LIN {X 0,Y 501.339,Z 1081.157,A -85,B 0,C 180,E1 23643.313,E2 23643.313} C_VEL
LIN {X 0,Y 503.042,Z 1063.83,A -85,B 0,C 180,E1 23641.19,E2 23641.19} C_VEL
LIN {X 0,Y 504.709,Z 1046.952,A -85,B 0,C 180,E1 23639.393,E2 23639.393} C_VEL
LIN {X 0,Y 506.659,Z 1027.452,A -85,B 0,C 180,E1 23637.597,E2 23637.597} C_VEL
LIN {X 0,Y 508.469,Z 1008.885,A -85,B 0,C 180,E1 23636.118,E2 23636.118} C_VEL
LIN {X 0,Y 510.36,Z 987.812,A -85,B 0,C 180,E1 23634.694,E2 23634.694} C_VEL
LIN {X 0,Y 512.134,Z 967.274,A -85,B 0,C 180,E1 23633.523,E2 23633.523} C_VEL
LIN {X 0,Y 513.653,Z 946.062,A -85,B 0,C 180,E1 23632.54,E2 23632.54} C_VEL
LIN {X 0,Y 515.046,Z 923.99,A -85,B 0,C 180,E1 23631.712,E2 23631.712} C_VEL
LIN {X 0,Y 516.104,Z 901.792,A -85,B 0,C 180,E1 23631.102,E2 23631.102} C_VEL
LIN {X 0,Y 516.884,Z 877.055,A -85,B 0,C 180,E1 23630.622,E2 23630.622} C_VEL
LIN {X 0,Y 520.36,Z 675.514,A -85,B 0,C 180,E1 23627.344,E2 23627.344} C_VEL
LIN {X 0,Y 522.211,Z 567.304,A -85,B 0,C 180,E1 23625.529,E2 23625.529} C_VEL
LIN {X 0,Y 521.353,Z 564.118,A -85,B 0,C 180,E1 23625.377,E2 23625.377} C_VEL
LIN {X 0,Y 506.181,Z 540.947,A -85,B 0,C 180,E1 23623.206,E2 23623.206} C_VEL
LIN {X 0,Y 500.368,Z 529.073,A -85,B 0,C 180,E1 23621.408,E2 23621.408} C_VEL
LIN {X 0,Y 498.57,Z 525.359,A -85,B 0,C 180,E1 23620.827,E2 23620.827} C_VEL
LIN {X 0,Y 496.912,Z 522.181,A -85,B 0,C 180,E1 23620.305,E2 23620.305} C_VEL
LIN {X 0,Y 496.727,Z 521.177,A -85,B 0,C 180,E1 23620.175,E2 23620.175} C_VEL
LIN {X 0,Y 496.731,Z 521.174,A -85,B 0,C 180,E1 23616.568,E2 23616.568} C_VEL
LIN {X 0,Y 496.77,Z 521.152,A -85,B 0,C 180,E1 23613.055,E2 23613.055} C_VEL
LIN {X 0,Y 496.742,Z 521.144,A -85,B 0,C 180,E1 23609.547,E2 23609.547} C_VEL
LIN {X 0,Y 496.741,Z 521.166,A -85,B 0,C 180,E1 23606.027,E2 23606.027} C_VEL
LIN {X 0,Y 496.765,Z 521.148,A -85,B 0,C 180,E1 23602.483,E2 23602.483} C_VEL
LIN {X 0,Y 496.759,Z 521.148,A -85,B 0,C 180,E1 23598.908,E2 23598.908} C_VEL
LIN {X 0,Y 496.747,Z 521.161,A -85,B 0,C 180,E1 23595.389,E2 23595.389} C_VEL
LIN {X 0,Y 496.76,Z 521.146,A -85,B 0,C 180,E1 23591.965,E2 23591.965} C_VEL
LIN {X 0,Y 496.766,Z 521.164,A -85,B 0,C 180,E1 23588.332,E2 23588.332} C_VEL
LIN {X 0,Y 496.756,Z 521.163,A -85,B 0,C 180,E1 23584.733,E2 23584.733} C_VEL
LIN {X 0,Y 496.765,Z 521.162,A -85,B 0,C 180,E1 23581.153,E2 23581.153} C_VEL
LIN {X 0,Y 496.749,Z 521.17,A -85,B 0,C 180,E1 23577.577,E2 23577.577} C_VEL
LIN {X 0,Y 496.767,Z 521.163,A -85,B 0,C 180,E1 23573.992,E2 23573.992} C_VEL
LIN {X 0,Y 496.764,Z 521.144,A -85,B 0,C 180,E1 23570.383,E2 23570.383} C_VEL
LIN {X 0,Y 496.739,Z 521.168,A -85,B 0,C 180,E1 23566.853,E2 23566.853} C_VEL
LIN {X 0,Y 496.756,Z 521.139,A -85,B 0,C 180,E1 23563.354,E2 23563.354} C_VEL
LIN {X 0,Y 496.765,Z 521.164,A -85,B 0,C 180,E1 23559.868,E2 23559.868} C_VEL
LIN {X 0,Y 496.722,Z 521.139,A -85,B 0,C 180,E1 23556.512,E2 23556.512} C_VEL
LIN {X 0,Y 496.769,Z 521.171,A -85,B 0,C 180,E1 23553.072,E2 23553.072} C_VEL
LIN {X 0,Y 496.728,Z 521.149,A -85,B 0,C 180,E1 23549.653,E2 23549.653} C_VEL
LIN {X 0,Y 496.717,Z 521.157,A -85,B 0,C 180,E1 23546.238,E2 23546.238} C_VEL
LIN {X 0,Y 496.767,Z 521.171,A -85,B 0,C 180,E1 23542.849,E2 23542.849} C_VEL
LIN {X 0,Y 496.704,Z 521.167,A -85,B 0,C 180,E1 23539.444,E2 23539.444} C_VEL
LIN {X 0,Y 496.719,Z 521.291,A -85,B 0,C 180,E1 23537.8,E2 23537.8} C_VEL
LIN {X 0,Y 497.882,Z 524.471,A -85,B 0,C 180,E1 23537.584,E2 23537.584} C_VEL
LIN {X 0,Y 500.714,Z 527.592,A -85,B 0,C 180,E1 23537.161,E2 23537.161} C_VEL
LIN {X 0,Y 503.416,Z 531.516,A -85,B 0,C 180,E1 23536.747,E2 23536.747} C_VEL
LIN {X 0,Y 515.125,Z 547.854,A -85,B 0,C 180,E1 23535.047,E2 23535.047} C_VEL
LIN {X 0,Y 522.101,Z 558.293,A -85,B 0,C 180,E1 23534.08,E2 23534.08} C_VEL
LIN {X 0,Y 521.82,Z 573.27,A -85,B 0,C 180,E1 23533.828,E2 23533.828} C_VEL
LIN {X 0,Y 520.938,Z 580.975,A -85,B 0,C 180,E1 23533.777,E2 23533.777} C_VEL
LIN {X 0,Y 516.065,Z 601.619,A -85,B 0,C 180,E1 23533.91,E2 23533.91} C_VEL
LIN {X 0,Y 515.408,Z 608.225,A -85,B 0,C 180,E1 23533.855,E2 23533.855} C_VEL
LIN {X 0,Y 511.275,Z 818.012,A -85,B 0,C 180,E1 23530.381,E2 23530.381} C_VEL
LIN {X 0,Y 510.22,Z 865.585,A -85,B 0,C 180,E1 23529.57,E2 23529.57} C_VEL
LIN {X 0,Y 509.144,Z 887.086,A -85,B 0,C 180,E1 23529.015,E2 23529.015} C_VEL
LIN {X 0,Y 507.847,Z 908.352,A -85,B 0,C 180,E1 23528.294,E2 23528.294} C_VEL
LIN {X 0,Y 506.128,Z 930.123,A -85,B 0,C 180,E1 23527.336,E2 23527.336} C_VEL
LIN {X 0,Y 504.269,Z 952.142,A -85,B 0,C 180,E1 23526.149,E2 23526.149} C_VEL
LIN {X 0,Y 502.401,Z 971.336,A -85,B 0,C 180,E1 23524.902,E2 23524.902} C_VEL
LIN {X 0,Y 500.276,Z 991.897,A -85,B 0,C 180,E1 23523.34,E2 23523.34} C_VEL
LIN {X 0,Y 498.327,Z 1010.198,A -85,B 0,C 180,E1 23521.709,E2 23521.709} C_VEL
LIN {X 0,Y 496.2,Z 1029.513,A -85,B 0,C 180,E1 23519.716,E2 23519.716} C_VEL
LIN {X 0,Y 494.437,Z 1046.319,A -85,B 0,C 180,E1 23517.718,E2 23517.718} C_VEL
LIN {X 0,Y 492.742,Z 1062.531,A -85,B 0,C 180,E1 23515.48,E2 23515.48} C_VEL
LIN {X 0,Y 491.262,Z 1078.098,A -85,B 0,C 180,E1 23513.003,E2 23513.003} C_VEL
LIN {X 0,Y 490.193,Z 1090.761,A -85,B 0,C 180,E1 23510.663,E2 23510.663} C_VEL
LIN {X 0,Y 489.317,Z 1102.656,A -85,B 0,C 180,E1 23508.095,E2 23508.095} C_VEL
LIN {X 0,Y 488.702,Z 1112.905,A -85,B 0,C 180,E1 23505.497,E2 23505.497} C_VEL
LIN {X 0,Y 488.285,Z 1121.274,A -85,B 0,C 180,E1 23502.897,E2 23502.897} C_VEL
LIN {X 0,Y 488.063,Z 1128.202,A -85,B 0,C 180,E1 23500.267,E2 23500.267} C_VEL
LIN {X 0,Y 487.966,Z 1133.176,A -85,B 0,C 180,E1 23497.773,E2 23497.773} C_VEL
LIN {X 0,Y 487.917,Z 1137.117,A -85,B 0,C 180,E1 23495.056,E2 23495.056} C_VEL
LIN {X 0,Y 487.91,Z 1139.232,A -85,B 0,C 180,E1 23492.467,E2 23492.467} C_VEL
LIN {X 0,Y 487.908,Z 1139.993,A -85,B 0,C 180,E1 23489.883,E2 23489.883} C_VEL
LIN {X 0,Y 487.904,Z 1139.148,A -85,B 0,C 180,E1 23487.299,E2 23487.299} C_VEL
LIN {X 0,Y 487.917,Z 1136.97,A -85,B 0,C 180,E1 23484.709,E2 23484.709} C_VEL
LIN {X 0,Y 487.97,Z 1133.127,A -85,B 0,C 180,E1 23482.109,E2 23482.109} C_VEL
LIN {X 0,Y 488.081,Z 1127.881,A -85,B 0,C 180,E1 23479.495,E2 23479.495} C_VEL
LIN {X 0,Y 488.313,Z 1120.835,A -85,B 0,C 180,E1 23476.863,E2 23476.863} C_VEL
LIN {X 0,Y 488.739,Z 1112.155,A -85,B 0,C 180,E1 23474.211,E2 23474.211} C_VEL
LIN {X 0,Y 489.361,Z 1102.001,A -85,B 0,C 180,E1 23471.66,E2 23471.66} C_VEL
LIN {X 0,Y 490.305,Z 1089.313,A -85,B 0,C 180,E1 23468.967,E2 23468.967} C_VEL
LIN {X 0,Y 491.452,Z 1076.174,A -85,B 0,C 180,E1 23466.572,E2 23466.572} C_VEL
LIN {X 0,Y 492.861,Z 1061.34,A -85,B 0,C 180,E1 23464.255,E2 23464.255} C_VEL
LIN {X 0,Y 494.567,Z 1044.991,A -85,B 0,C 180,E1 23462.029,E2 23462.029} C_VEL
LIN {X 0,Y 496.302,Z 1028.605,A -85,B 0,C 180,E1 23460.091,E2 23460.091} C_VEL
LIN {X 0,Y 498.378,Z 1009.706,A -85,B 0,C 180,E1 23458.154,E2 23458.154} C_VEL
LIN {X 0,Y 500.334,Z 991.393,A -85,B 0,C 180,E1 23456.526,E2 23456.526} C_VEL
LIN {X 0,Y 502.374,Z 971.61,A -85,B 0,C 180,E1 23455.027,E2 23455.027} C_VEL
LIN {X 0,Y 504.24,Z 952.427,A -85,B 0,C 180,E1 23453.779,E2 23453.779} C_VEL
LIN {X 0,Y 506.064,Z 930.957,A -85,B 0,C 180,E1 23452.615,E2 23452.615} C_VEL
LIN {X 0,Y 507.833,Z 908.532,A -85,B 0,C 180,E1 23451.623,E2 23451.623} C_VEL
LIN {X 0,Y 509.134,Z 887.292,A -85,B 0,C 180,E1 23450.901,E2 23450.901} C_VEL
LIN {X 0,Y 510.198,Z 866.05,A -85,B 0,C 180,E1 23450.351,E2 23450.351} C_VEL
LIN {X 0,Y 511.17,Z 823.523,A -85,B 0,C 180,E1 23449.619,E2 23449.619} C_VEL
LIN {X 0,Y 515.352,Z 611.14,A -85,B 0,C 180,E1 23446.104,E2 23446.104} C_VEL
LIN {X 0,Y 516.192,Z 561.548,A -85,B 0,C 180,E1 23445.247,E2 23445.247} C_VEL
LIN {X 0,Y 503.138,Z 542.859,A -85,B 0,C 180,E1 23443.361,E2 23443.361} C_VEL
LIN {X 0,Y 495.758,Z 532.811,A -85,B 0,C 180,E1 23442.23,E2 23442.23} C_VEL
LIN {X 0,Y 493.019,Z 529.057,A -85,B 0,C 180,E1 23441.795,E2 23441.795} C_VEL
LIN {X 0,Y 492.07,Z 527.668,A -85,B 0,C 180,E1 23441.64,E2 23441.64} C_VEL
LIN {X 0,Y 489.619,Z 524.782,A -85,B 0,C 180,E1 23441.25,E2 23441.25} C_VEL
LIN {X 0,Y 488.798,Z 522.162,A -85,B 0,C 180,E1 23441.07,E2 23441.07} C_VEL
LIN {X 0,Y 488.779,Z 522.154,A -85,B 0,C 180,E1 23437.708,E2 23437.708} C_VEL
LIN {X 0,Y 488.767,Z 522.136,A -85,B 0,C 180,E1 23434.233,E2 23434.233} C_VEL
LIN {X 0,Y 488.832,Z 522.142,A -85,B 0,C 180,E1 23430.754,E2 23430.754} C_VEL
LIN {X 0,Y 488.792,Z 522.155,A -85,B 0,C 180,E1 23427.272,E2 23427.272} C_VEL
LIN {X 0,Y 488.782,Z 522.128,A -85,B 0,C 180,E1 23423.765,E2 23423.765} C_VEL
LIN {X 0,Y 488.835,Z 522.157,A -85,B 0,C 180,E1 23420.348,E2 23420.348} C_VEL
LIN {X 0,Y 488.8,Z 522.124,A -85,B 0,C 180,E1 23416.801,E2 23416.801} C_VEL
LIN {X 0,Y 488.799,Z 522.158,A -85,B 0,C 180,E1 23413.244,E2 23413.244} C_VEL
LIN {X 0,Y 488.829,Z 522.155,A -85,B 0,C 180,E1 23409.775,E2 23409.775} C_VEL
LIN {X 0,Y 488.821,Z 522.161,A -85,B 0,C 180,E1 23406.224,E2 23406.224} C_VEL
LIN {X 0,Y 488.806,Z 522.159,A -85,B 0,C 180,E1 23402.58,E2 23402.58} C_VEL
LIN {X 0,Y 488.829,Z 522.154,A -85,B 0,C 180,E1 23399.063,E2 23399.063} C_VEL
LIN {X 0,Y 488.822,Z 522.157,A -85,B 0,C 180,E1 23395.425,E2 23395.425} C_VEL
LIN {X 0,Y 488.819,Z 522.159,A -85,B 0,C 180,E1 23391.887,E2 23391.887} C_VEL
LIN {X 0,Y 488.823,Z 522.122,A -85,B 0,C 180,E1 23388.317,E2 23388.317} C_VEL
LIN {X 0,Y 488.811,Z 522.155,A -85,B 0,C 180,E1 23384.822,E2 23384.822} C_VEL
LIN {X 0,Y 488.825,Z 522.13,A -85,B 0,C 180,E1 23381.269,E2 23381.269} C_VEL
LIN {X 0,Y 488.83,Z 522.144,A -85,B 0,C 180,E1 23377.639,E2 23377.639} C_VEL
LIN {X 0,Y 488.803,Z 522.159,A -85,B 0,C 180,E1 23374.04,E2 23374.04} C_VEL
LIN {X 0,Y 488.802,Z 522.135,A -85,B 0,C 180,E1 23370.383,E2 23370.383} C_VEL
LIN {X 0,Y 488.831,Z 522.137,A -85,B 0,C 180,E1 23366.899,E2 23366.899} C_VEL
LIN {X 0,Y 488.792,Z 522.161,A -85,B 0,C 180,E1 23363.469,E2 23363.469} C_VEL
LIN {X 0,Y 488.861,Z 522.355,A -85,B 0,C 180,E1 23360.759,E2 23360.759} C_VEL
LIN {X 0,Y 490.363,Z 525.981,A -85,B 0,C 180,E1 23360.19,E2 23360.19} C_VEL
LIN {X 0,Y 491.426,Z 528.1,A -85,B 0,C 180,E1 23359.837,E2 23359.837} C_VEL
LIN {X 0,Y 495.467,Z 535.911,A -85,B 0,C 180,E1 23358.555,E2 23358.555} C_VEL
LIN {X 0,Y 498.071,Z 541.152,A -85,B 0,C 180,E1 23357.783,E2 23357.783} C_VEL
LIN {X 0,Y 511.268,Z 561.075,A -85,B 0,C 180,E1 23355.799,E2 23355.799} C_VEL
LIN {X 0,Y 516.559,Z 569.744,A -85,B 0,C 180,E1 23355.037,E2 23355.037} C_VEL
LIN {X 0,Y 513.282,Z 735.937,A -85,B 0,C 180,E1 23352.257,E2 23352.257} C_VEL
LIN {X 0,Y 510.262,Z 891.967,A -85,B 0,C 180,E1 23349.679,E2 23349.679} C_VEL
LIN {X 0,Y 509.215,Z 914.865,A -85,B 0,C 180,E1 23349.119,E2 23349.119} C_VEL
LIN {X 0,Y 508.04,Z 934.757,A -85,B 0,C 180,E1 23348.465,E2 23348.465} C_VEL
LIN {X 0,Y 506.385,Z 957.093,A -85,B 0,C 180,E1 23347.527,E2 23347.527} C_VEL
LIN {X 0,Y 504.587,Z 978.468,A -85,B 0,C 180,E1 23346.411,E2 23346.411} C_VEL
LIN {X 0,Y 502.614,Z 999.226,A -85,B 0,C 180,E1 23345.093,E2 23345.093} C_VEL
LIN {X 0,Y 500.642,Z 1018.623,A -85,B 0,C 180,E1 23343.656,E2 23343.656} C_VEL
LIN {X 0,Y 498.56,Z 1037.927,A -85,B 0,C 180,E1 23341.968,E2 23341.968} C_VEL
LIN {X 0,Y 496.548,Z 1056.565,A -85,B 0,C 180,E1 23340.092,E2 23340.092} C_VEL
LIN {X 0,Y 494.748,Z 1073.124,A -85,B 0,C 180,E1 23338.157,E2 23338.157} C_VEL
LIN {X 0,Y 492.965,Z 1090.295,A -85,B 0,C 180,E1 23335.854,E2 23335.854} C_VEL
LIN {X 0,Y 491.518,Z 1105.507,A -85,B 0,C 180,E1 23333.497,E2 23333.497} C_VEL
LIN {X 0,Y 490.322,Z 1119.085,A -85,B 0,C 180,E1 23331.032,E2 23331.032} C_VEL
LIN {X 0,Y 489.407,Z 1131.29,A -85,B 0,C 180,E1 23328.461,E2 23328.461} C_VEL
LIN {X 0,Y 488.785,Z 1141.067,A -85,B 0,C 180,E1 23326.031,E2 23326.031} C_VEL
LIN {X 0,Y 488.334,Z 1150.349,A -85,B 0,C 180,E1 23323.257,E2 23323.257} C_VEL
LIN {X 0,Y 488.107,Z 1157.169,A -85,B 0,C 180,E1 23320.743,E2 23320.743} C_VEL
LIN {X 0,Y 487.975,Z 1162.635,A -85,B 0,C 180,E1 23318.128,E2 23318.128} C_VEL
LIN {X 0,Y 487.906,Z 1166.438,A -85,B 0,C 180,E1 23315.645,E2 23315.645} C_VEL
LIN {X 0,Y 487.89,Z 1168.986,A -85,B 0,C 180,E1 23312.937,E2 23312.937} C_VEL
LIN {X 0,Y 487.885,Z 1169.895,A -85,B 0,C 180,E1 23310.587,E2 23310.587} C_VEL
LIN {X 0,Y 487.914,Z 1169.392,A -85,B 0,C 180,E1 23307.768,E2 23307.768} C_VEL
LIN {X 0,Y 487.909,Z 1167.501,A -85,B 0,C 180,E1 23305.298,E2 23305.298} C_VEL
LIN {X 0,Y 487.933,Z 1163.874,A -85,B 0,C 180,E1 23302.582,E2 23302.582} C_VEL
LIN {X 0,Y 488.014,Z 1159.573,A -85,B 0,C 180,E1 23300.328,E2 23300.328} C_VEL
LIN {X 0,Y 488.213,Z 1153.516,A -85,B 0,C 180,E1 23297.822,E2 23297.822} C_VEL
LIN {X 0,Y 488.562,Z 1145.341,A -85,B 0,C 180,E1 23295.178,E2 23295.178} C_VEL
LIN {X 0,Y 489.13,Z 1135.417,A -85,B 0,C 180,E1 23292.513,E2 23292.513} C_VEL
LIN {X 0,Y 489.891,Z 1124.575,A -85,B 0,C 180,E1 23290.071,E2 23290.071} C_VEL
LIN {X 0,Y 490.992,Z 1111.15,A -85,B 0,C 180,E1 23287.49,E2 23287.49} C_VEL
LIN {X 0,Y 492.316,Z 1097.011,A -85,B 0,C 180,E1 23285.14,E2 23285.14} C_VEL
LIN {X 0,Y 493.871,Z 1081.33,A -85,B 0,C 180,E1 23282.901,E2 23282.901} C_VEL
LIN {X 0,Y 495.764,Z 1063.774,A -85,B 0,C 180,E1 23280.72,E2 23280.72} C_VEL
LIN {X 0,Y 497.616,Z 1046.551,A -85,B 0,C 180,E1 23278.865,E2 23278.865} C_VEL
LIN {X 0,Y 499.765,Z 1026.775,A -85,B 0,C 180,E1 23277.031,E2 23277.031} C_VEL
LIN {X 0,Y 501.819,Z 1007.26,A -85,B 0,C 180,E1 23275.468,E2 23275.468} C_VEL
LIN {X 0,Y 503.804,Z 986.803,A -85,B 0,C 180,E1 23274.094,E2 23274.094} C_VEL
LIN {X 0,Y 505.708,Z 966.071,A -85,B 0,C 180,E1 23272.912,E2 23272.912} C_VEL
LIN {X 0,Y 507.292,Z 945.156,A -85,B 0,C 180,E1 23271.944,E2 23271.944} C_VEL
LIN {X 0,Y 508.798,Z 922.523,A -85,B 0,C 180,E1 23271.108,E2 23271.108} C_VEL
LIN {X 0,Y 509.869,Z 901.392,A -85,B 0,C 180,E1 23270.529,E2 23270.529} C_VEL
LIN {X 0,Y 510.697,Z 876.242,A -85,B 0,C 180,E1 23270.041,E2 23270.041} C_VEL
LIN {X 0,Y 514.468,Z 675.084,A -85,B 0,C 180,E1 23266.734,E2 23266.734} C_VEL
LIN {X 0,Y 516.46,Z 569.215,A -85,B 0,C 180,E1 23264.942,E2 23264.942} C_VEL
LIN {X 0,Y 501.454,Z 546.105,A -85,B 0,C 180,E1 23262.74,E2 23262.74} C_VEL
LIN {X 0,Y 497.653,Z 540.451,A -85,B 0,C 180,E1 23262.148,E2 23262.148} C_VEL
LIN {X 0,Y 492.496,Z 530.229,A -85,B 0,C 180,E1 23260.515,E2 23260.515} C_VEL
LIN {X 0,Y 490.353,Z 525.974,A -85,B 0,C 180,E1 23259.811,E2 23259.811} C_VEL
LIN {X 0,Y 488.857,Z 522.324,A -85,B 0,C 180,E1 23259.241,E2 23259.241} C_VEL
LIN {X 0,Y 488.808,Z 522.153,A -85,B 0,C 180,E1 23255.701,E2 23255.701} C_VEL
LIN {X 0,Y 488.791,Z 522.159,A -85,B 0,C 180,E1 23252.126,E2 23252.126} C_VEL
LIN {X 0,Y 488.829,Z 522.13,A -85,B 0,C 180,E1 23248.595,E2 23248.595} C_VEL
LIN {X 0,Y 488.825,Z 522.135,A -85,B 0,C 180,E1 23245.023,E2 23245.023} C_VEL
LIN {X 0,Y 488.803,Z 522.152,A -85,B 0,C 180,E1 23241.452,E2 23241.452} C_VEL
LIN {X 0,Y 488.818,Z 522.121,A -85,B 0,C 180,E1 23237.867,E2 23237.867} C_VEL
LIN {X 0,Y 488.825,Z 522.159,A -85,B 0,C 180,E1 23234.329,E2 23234.329} C_VEL
LIN {X 0,Y 488.816,Z 522.123,A -85,B 0,C 180,E1 23230.727,E2 23230.727} C_VEL
LIN {X 0,Y 488.822,Z 522.156,A -85,B 0,C 180,E1 23227.167,E2 23227.167} C_VEL
LIN {X 0,Y 488.815,Z 522.157,A -85,B 0,C 180,E1 23223.635,E2 23223.635} C_VEL
LIN {X 0,Y 488.827,Z 522.159,A -85,B 0,C 180,E1 23220,E2 23220} C_VEL
LIN {X 0,Y 488.824,Z 522.158,A -85,B 0,C 180,E1 23216.364,E2 23216.364} C_VEL
LIN {X 0,Y 488.825,Z 522.155,A -85,B 0,C 180,E1 23212.714,E2 23212.714} C_VEL
LIN {X 0,Y 488.798,Z 522.125,A -85,B 0,C 180,E1 23209.074,E2 23209.074} C_VEL
LIN {X 0,Y 488.832,Z 522.158,A -85,B 0,C 180,E1 23205.55,E2 23205.55} C_VEL
LIN {X 0,Y 488.827,Z 522.122,A -85,B 0,C 180,E1 23201.886,E2 23201.886} C_VEL
LIN {X 0,Y 488.792,Z 522.156,A -85,B 0,C 180,E1 23198.395,E2 23198.395} C_VEL
LIN {X 0,Y 488.799,Z 522.14,A -85,B 0,C 180,E1 23194.819,E2 23194.819} C_VEL
LIN {X 0,Y 488.834,Z 522.134,A -85,B 0,C 180,E1 23191.34,E2 23191.34} C_VEL
LIN {X 0,Y 488.779,Z 522.162,A -85,B 0,C 180,E1 23187.868,E2 23187.868} C_VEL
LIN {X 0,Y 488.783,Z 522.143,A -85,B 0,C 180,E1 23184.303,E2 23184.303} C_VEL
LIN {X 0,Y 488.809,Z 522.134,A -85,B 0,C 180,E1 23180.949,E2 23180.949} C_VEL
LIN {X 0,Y 488.831,Z 522.299,A -85,B 0,C 180,E1 23178.818,E2 23178.818} C_VEL
LIN {X 0,Y 490.064,Z 525.535,A -85,B 0,C 180,E1 23178.581,E2 23178.581} C_VEL
LIN {X 0,Y 492.832,Z 528.661,A -85,B 0,C 180,E1 23178.147,E2 23178.147} C_VEL
LIN {X 0,Y 495.553,Z 532.605,A -85,B 0,C 180,E1 23177.709,E2 23177.709} C_VEL
LIN {X 0,Y 497.132,Z 534.605,A -85,B 0,C 180,E1 23177.465,E2 23177.465} C_VEL
LIN {X 0,Y 510.465,Z 553.132,A -85,B 0,C 180,E1 23175.475,E2 23175.475} C_VEL
LIN {X 0,Y 516.314,Z 562.022,A -85,B 0,C 180,E1 23174.64,E2 23174.64} C_VEL
LIN {X 0,Y 515.408,Z 608.225,A -85,B 0,C 180,E1 23173.855,E2 23173.855} C_VEL
LIN {X 0,Y 514.536,Z 615.928,A -85,B 0,C 180,E1 23173.803,E2 23173.803} C_VEL
LIN {X 0,Y 509.557,Z 636.554,A -85,B 0,C 180,E1 23173.949,E2 23173.949} C_VEL
LIN {X 0,Y 508.877,Z 643.162,A -85,B 0,C 180,E1 23173.896,E2 23173.896} C_VEL
LIN {X 0,Y 504.713,Z 842.961,A -85,B 0,C 180,E1 23170.563,E2 23170.563} C_VEL
LIN {X 0,Y 503.803,Z 871.088,A -85,B 0,C 180,E1 23170.027,E2 23170.027} C_VEL
LIN {X 0,Y 502.74,Z 890.849,A -85,B 0,C 180,E1 23169.487,E2 23169.487} C_VEL
LIN {X 0,Y 501.099,Z 913.862,A -85,B 0,C 180,E1 23168.649,E2 23168.649} C_VEL
LIN {X 0,Y 499.365,Z 934.763,A -85,B 0,C 180,E1 23167.68,E2 23167.68} C_VEL
LIN {X 0,Y 497.285,Z 956.054,A -85,B 0,C 180,E1 23166.462,E2 23166.462} C_VEL
LIN {X 0,Y 495.126,Z 976.727,A -85,B 0,C 180,E1 23165.067,E2 23165.067} C_VEL
LIN {X 0,Y 492.895,Z 996.298,A -85,B 0,C 180,E1 23163.489,E2 23163.489} C_VEL
LIN {X 0,Y 490.692,Z 1015.331,A -85,B 0,C 180,E1 23161.717,E2 23161.717} C_VEL
LIN {X 0,Y 488.602,Z 1032.911,A -85,B 0,C 180,E1 23159.812,E2 23159.812} C_VEL
LIN {X 0,Y 486.55,Z 1050.552,A -85,B 0,C 180,E1 23157.607,E2 23157.607} C_VEL
LIN {X 0,Y 484.884,Z 1065.915,A -85,B 0,C 180,E1 23155.399,E2 23155.399} C_VEL
LIN {X 0,Y 483.397,Z 1080.22,A -85,B 0,C 180,E1 23153.009,E2 23153.009} C_VEL
LIN {X 0,Y 482.221,Z 1093.21,A -85,B 0,C 180,E1 23150.513,E2 23150.513} C_VEL
LIN {X 0,Y 481.354,Z 1104.202,A -85,B 0,C 180,E1 23148.029,E2 23148.029} C_VEL
LIN {X 0,Y 480.667,Z 1114.787,A -85,B 0,C 180,E1 23145.195,E2 23145.195} C_VEL
LIN {X 0,Y 480.268,Z 1122.688,A -85,B 0,C 180,E1 23142.627,E2 23142.627} C_VEL
LIN {X 0,Y 480.035,Z 1129.224,A -85,B 0,C 180,E1 23139.956,E2 23139.956} C_VEL
LIN {X 0,Y 479.957,Z 1133.59,A -85,B 0,C 180,E1 23137.662,E2 23137.662} C_VEL
LIN {X 0,Y 479.915,Z 1137.344,A -85,B 0,C 180,E1 23134.9,E2 23134.9} C_VEL
LIN {X 0,Y 479.912,Z 1139.3,A -85,B 0,C 180,E1 23132.388,E2 23132.388} C_VEL
LIN {X 0,Y 479.892,Z 1139.948,A -85,B 0,C 180,E1 23129.642,E2 23129.642} C_VEL
LIN {X 0,Y 479.902,Z 1139.148,A -85,B 0,C 180,E1 23127.254,E2 23127.254} C_VEL
LIN {X 0,Y 479.917,Z 1136.969,A -85,B 0,C 180,E1 23124.621,E2 23124.621} C_VEL
LIN {X 0,Y 479.978,Z 1133.126,A -85,B 0,C 180,E1 23121.977,E2 23121.977} C_VEL
LIN {X 0,Y 480.107,Z 1127.879,A -85,B 0,C 180,E1 23119.319,E2 23119.319} C_VEL
LIN {X 0,Y 480.362,Z 1120.832,A -85,B 0,C 180,E1 23116.642,E2 23116.642} C_VEL
LIN {X 0,Y 480.825,Z 1112.15,A -85,B 0,C 180,E1 23113.945,E2 23113.945} C_VEL
LIN {X 0,Y 481.477,Z 1102.511,A -85,B 0,C 180,E1 23111.475,E2 23111.475} C_VEL
LIN {X 0,Y 482.503,Z 1089.942,A -85,B 0,C 180,E1 23108.738,E2 23108.738} C_VEL
LIN {X 0,Y 483.71,Z 1077.184,A -85,B 0,C 180,E1 23106.359,E2 23106.359} C_VEL
LIN {X 0,Y 485.274,Z 1062.091,A -85,B 0,C 180,E1 23103.94,E2 23103.94} C_VEL
LIN {X 0,Y 487.11,Z 1045.998,A -85,B 0,C 180,E1 23101.696,E2 23101.696} C_VEL
LIN {X 0,Y 489.041,Z 1029.151,A -85,B 0,C 180,E1 23099.669,E2 23099.669} C_VEL
LIN {X 0,Y 491.379,Z 1009.372,A -85,B 0,C 180,E1 23097.612,E2 23097.612} C_VEL
LIN {X 0,Y 493.524,Z 990.907,A -85,B 0,C 180,E1 23095.957,E2 23095.957} C_VEL
LIN {X 0,Y 495.758,Z 970.694,A -85,B 0,C 180,E1 23094.419,E2 23094.419} C_VEL
LIN {X 0,Y 497.881,Z 950.461,A -85,B 0,C 180,E1 23093.097,E2 23093.097} C_VEL
LIN {X 0,Y 499.808,Z 929.406,A -85,B 0,C 180,E1 23091.965,E2 23091.965} C_VEL
LIN {X 0,Y 501.666,Z 907.09,A -85,B 0,C 180,E1 23090.989,E2 23090.989} C_VEL
LIN {X 0,Y 502.975,Z 886.817,A -85,B 0,C 180,E1 23090.302,E2 23090.302} C_VEL
LIN {X 0,Y 504.111,Z 865.028,A -85,B 0,C 180,E1 23089.742,E2 23089.742} C_VEL
LIN {X 0,Y 505.544,Z 801.78,A -85,B 0,C 180,E1 23088.667,E2 23088.667} C_VEL
LIN {X 0,Y 510.059,Z 589.597,A -85,B 0,C 180,E1 23085.106,E2 23085.106} C_VEL
LIN {X 0,Y 510.416,Z 565.256,A -85,B 0,C 180,E1 23084.669,E2 23084.669} C_VEL
LIN {X 0,Y 498.717,Z 548.51,A -85,B 0,C 180,E1 23082.934,E2 23082.934} C_VEL
LIN {X 0,Y 491.702,Z 538.917,A -85,B 0,C 180,E1 23081.834,E2 23081.834} C_VEL
LIN {X 0,Y 487.888,Z 533.76,A -85,B 0,C 180,E1 23081.214,E2 23081.214} C_VEL
LIN {X 0,Y 485.077,Z 529.758,A -85,B 0,C 180,E1 23080.741,E2 23080.741} C_VEL
LIN {X 0,Y 483.973,Z 528.567,A -85,B 0,C 180,E1 23080.561,E2 23080.561} C_VEL
LIN {X 0,Y 481.652,Z 525.825,A -85,B 0,C 180,E1 23080.172,E2 23080.172} C_VEL
LIN {X 0,Y 480.826,Z 523.131,A -85,B 0,C 180,E1 23079.983,E2 23079.983} C_VEL
LIN {X 0,Y 480.829,Z 523.152,A -85,B 0,C 180,E1 23076.345,E2 23076.345} C_VEL
LIN {X 0,Y 480.885,Z 523.137,A -85,B 0,C 180,E1 23072.86,E2 23072.86} C_VEL
LIN {X 0,Y 480.846,Z 523.119,A -85,B 0,C 180,E1 23069.389,E2 23069.389} C_VEL
LIN {X 0,Y 480.843,Z 523.149,A -85,B 0,C 180,E1 23065.76,E2 23065.76} C_VEL
LIN {X 0,Y 480.89,Z 523.122,A -85,B 0,C 180,E1 23062.236,E2 23062.236} C_VEL
LIN {X 0,Y 480.876,Z 523.128,A -85,B 0,C 180,E1 23058.675,E2 23058.675} C_VEL
LIN {X 0,Y 480.853,Z 523.138,A -85,B 0,C 180,E1 23055.065,E2 23055.065} C_VEL
LIN {X 0,Y 480.88,Z 523.14,A -85,B 0,C 180,E1 23051.514,E2 23051.514} C_VEL
LIN {X 0,Y 480.89,Z 523.14,A -85,B 0,C 180,E1 23047.888,E2 23047.888} C_VEL
LIN {X 0,Y 480.873,Z 523.14,A -85,B 0,C 180,E1 23044.293,E2 23044.293} C_VEL
LIN {X 0,Y 480.874,Z 523.136,A -85,B 0,C 180,E1 23040.715,E2 23040.715} C_VEL
LIN {X 0,Y 480.883,Z 523.139,A -85,B 0,C 180,E1 23037.14,E2 23037.14} C_VEL
LIN {X 0,Y 480.886,Z 523.14,A -85,B 0,C 180,E1 23033.434,E2 23033.434} C_VEL
LIN {X 0,Y 480.878,Z 523.118,A -85,B 0,C 180,E1 23029.821,E2 23029.821} C_VEL
LIN {X 0,Y 480.892,Z 523.141,A -85,B 0,C 180,E1 23026.162,E2 23026.162} C_VEL
LIN {X 0,Y 480.866,Z 523.112,A -85,B 0,C 180,E1 23022.578,E2 23022.578} C_VEL
LIN {X 0,Y 480.884,Z 523.148,A -85,B 0,C 180,E1 23018.918,E2 23018.918} C_VEL
LIN {X 0,Y 480.888,Z 523.121,A -85,B 0,C 180,E1 23015.297,E2 23015.297} C_VEL
LIN {X 0,Y 480.869,Z 523.126,A -85,B 0,C 180,E1 23011.701,E2 23011.701} C_VEL
LIN {X 0,Y 480.856,Z 523.149,A -85,B 0,C 180,E1 23008.12,E2 23008.12} C_VEL
LIN {X 0,Y 480.884,Z 523.135,A -85,B 0,C 180,E1 23004.543,E2 23004.543} C_VEL
LIN {X 0,Y 480.846,Z 523.131,A -85,B 0,C 180,E1 23001.814,E2 23001.814} C_VEL
LIN {X 0,Y 481.866,Z 526.149,A -85,B 0,C 180,E1 23001.35,E2 23001.35} C_VEL
LIN {X 0,Y 483.39,Z 528.554,A -85,B 0,C 180,E1 23000.886,E2 23000.886} C_VEL
LIN {X 0,Y 489.618,Z 540.648,A -85,B 0,C 180,E1 22998.886,E2 22998.886} C_VEL
LIN {X 0,Y 504.715,Z 563.364,A -85,B 0,C 180,E1 22996.516,E2 22996.516} C_VEL
LIN {X 0,Y 510.835,Z 573.306,A -85,B 0,C 180,E1 22995.608,E2 22995.608} C_VEL
LIN {X 0,Y 506.828,Z 762.387,A -85,B 0,C 180,E1 22992.42,E2 22992.42} C_VEL
LIN {X 0,Y 504.081,Z 891.906,A -85,B 0,C 180,E1 22990.259,E2 22990.259} C_VEL
LIN {X 0,Y 502.95,Z 914.763,A -85,B 0,C 180,E1 22989.694,E2 22989.694} C_VEL
LIN {X 0,Y 501.656,Z 935.178,A -85,B 0,C 180,E1 22989.016,E2 22989.016} C_VEL
LIN {X 0,Y 499.821,Z 958.146,A -85,B 0,C 180,E1 22988.034,E2 22988.034} C_VEL
LIN {X 0,Y 497.919,Z 979.647,A -85,B 0,C 180,E1 22986.9,E2 22986.9} C_VEL
LIN {X 0,Y 495.819,Z 1000.123,A -85,B 0,C 180,E1 22985.576,E2 22985.576} C_VEL
LIN {X 0,Y 493.621,Z 1020.17,A -85,B 0,C 180,E1 22984.061,E2 22984.061} C_VEL
LIN {X 0,Y 491.391,Z 1039.26,A -85,B 0,C 180,E1 22982.353,E2 22982.353} C_VEL
LIN {X 0,Y 489.088,Z 1058.783,A -85,B 0,C 180,E1 22980.328,E2 22980.328} C_VEL
LIN {X 0,Y 487.195,Z 1075.15,A -85,B 0,C 180,E1 22978.366,E2 22978.366} C_VEL
LIN {X 0,Y 485.378,Z 1091.139,A -85,B 0,C 180,E1 22976.157,E2 22976.157} C_VEL
LIN {X 0,Y 483.813,Z 1106.228,A -85,B 0,C 180,E1 22973.765,E2 22973.765} C_VEL
LIN {X 0,Y 482.57,Z 1119.083,A -85,B 0,C 180,E1 22971.387,E2 22971.387} C_VEL
LIN {X 0,Y 481.56,Z 1131.291,A -85,B 0,C 180,E1 22968.773,E2 22968.773} C_VEL
LIN {X 0,Y 480.878,Z 1141.066,A -85,B 0,C 180,E1 22966.302,E2 22966.302} C_VEL
LIN {X 0,Y 480.379,Z 1150.349,A -85,B 0,C 180,E1 22963.48,E2 22963.48} C_VEL
LIN {X 0,Y 480.127,Z 1157.169,A -85,B 0,C 180,E1 22960.924,E2 22960.924} C_VEL
LIN {X 0,Y 479.98,Z 1162.635,A -85,B 0,C 180,E1 22958.264,E2 22958.264} C_VEL
LIN {X 0,Y 479.907,Z 1166.438,A -85,B 0,C 180,E1 22955.739,E2 22955.739} C_VEL
LIN {X 0,Y 479.889,Z 1168.986,A -85,B 0,C 180,E1 22952.986,E2 22952.986} C_VEL
LIN {X 0,Y 479.884,Z 1169.895,A -85,B 0,C 180,E1 22950.597,E2 22950.597} C_VEL
LIN {X 0,Y 479.914,Z 1169.392,A -85,B 0,C 180,E1 22947.731,E2 22947.731} C_VEL
LIN {X 0,Y 479.91,Z 1167.501,A -85,B 0,C 180,E1 22945.219,E2 22945.219} C_VEL
LIN {X 0,Y 479.943,Z 1163.874,A -85,B 0,C 180,E1 22942.458,E2 22942.458} C_VEL
LIN {X 0,Y 480.028,Z 1159.507,A -85,B 0,C 180,E1 22940.134,E2 22940.134} C_VEL
LIN {X 0,Y 480.255,Z 1153.171,A -85,B 0,C 180,E1 22937.495,E2 22937.495} C_VEL
LIN {X 0,Y 480.636,Z 1145.34,A -85,B 0,C 180,E1 22934.927,E2 22934.927} C_VEL
LIN {X 0,Y 481.267,Z 1135.416,A -85,B 0,C 180,E1 22932.217,E2 22932.217} C_VEL
LIN {X 0,Y 482.101,Z 1124.575,A -85,B 0,C 180,E1 22929.735,E2 22929.735} C_VEL
LIN {X 0,Y 483.31,Z 1111.148,A -85,B 0,C 180,E1 22927.112,E2 22927.112} C_VEL
LIN {X 0,Y 484.765,Z 1097.013,A -85,B 0,C 180,E1 22924.725,E2 22924.725} C_VEL
LIN {X 0,Y 486.457,Z 1081.328,A -85,B 0,C 180,E1 22922.453,E2 22922.453} C_VEL
LIN {X 0,Y 488.452,Z 1064.328,A -85,B 0,C 180,E1 22920.305,E2 22920.305} C_VEL
LIN {X 0,Y 490.425,Z 1047.391,A -85,B 0,C 180,E1 22918.451,E2 22918.451} C_VEL
LIN {X 0,Y 492.764,Z 1027.507,A -85,B 0,C 180,E1 22916.571,E2 22916.571} C_VEL
LIN {X 0,Y 494.864,Z 1008.879,A -85,B 0,C 180,E1 22915.053,E2 22915.053} C_VEL
LIN {X 0,Y 496.993,Z 988.81,A -85,B 0,C 180,E1 22913.666,E2 22913.666} C_VEL
LIN {X 0,Y 498.886,Z 969.272,A -85,B 0,C 180,E1 22912.528,E2 22912.528} C_VEL
LIN {X 0,Y 500.735,Z 947.084,A -85,B 0,C 180,E1 22911.464,E2 22911.464} C_VEL
LIN {X 0,Y 502.305,Z 925.39,A -85,B 0,C 180,E1 22910.631,E2 22910.631} C_VEL
LIN {X 0,Y 503.58,Z 902.883,A -85,B 0,C 180,E1 22909.989,E2 22909.989} C_VEL
LIN {X 0,Y 504.483,Z 879.641,A -85,B 0,C 180,E1 22909.515,E2 22909.515} C_VEL
LIN {X 0,Y 508.542,Z 678.812,A -85,B 0,C 180,E1 22906.179,E2 22906.179} C_VEL
LIN {X 0,Y 510.672,Z 572.789,A -85,B 0,C 180,E1 22904.363,E2 22904.363} C_VEL
LIN {X 0,Y 496.157,Z 550.277,A -85,B 0,C 180,E1 22902.168,E2 22902.168} C_VEL
LIN {X 0,Y 489.059,Z 539.882,A -85,B 0,C 180,E1 22901.015,E2 22901.015} C_VEL
LIN {X 0,Y 484.254,Z 530.592,A -85,B 0,C 180,E1 22899.446,E2 22899.446} C_VEL
LIN {X 0,Y 483.081,Z 527.74,A -85,B 0,C 180,E1 22898.991,E2 22898.991} C_VEL
LIN {X 0,Y 481.2,Z 524.712,A -85,B 0,C 180,E1 22898.409,E2 22898.409} C_VEL
LIN {X 0,Y 480.848,Z 523.154,A -85,B 0,C 180,E1 22898.186,E2 22898.186} C_VEL
LIN {X 0,Y 480.859,Z 523.122,A -85,B 0,C 180,E1 22894.571,E2 22894.571} C_VEL
LIN {X 0,Y 480.894,Z 523.138,A -85,B 0,C 180,E1 22891.039,E2 22891.039} C_VEL
LIN {X 0,Y 480.866,Z 523.136,A -85,B 0,C 180,E1 22887.49,E2 22887.49} C_VEL
LIN {X 0,Y 480.862,Z 523.111,A -85,B 0,C 180,E1 22883.92,E2 22883.92} C_VEL
LIN {X 0,Y 480.89,Z 523.143,A -85,B 0,C 180,E1 22880.444,E2 22880.444} C_VEL
LIN {X 0,Y 480.883,Z 523.111,A -85,B 0,C 180,E1 22876.798,E2 22876.798} C_VEL
LIN {X 0,Y 480.874,Z 523.146,A -85,B 0,C 180,E1 22873.221,E2 22873.221} C_VEL
LIN {X 0,Y 480.886,Z 523.122,A -85,B 0,C 180,E1 22869.575,E2 22869.575} C_VEL
LIN {X 0,Y 480.879,Z 523.138,A -85,B 0,C 180,E1 22865.967,E2 22865.967} C_VEL
LIN {X 0,Y 480.884,Z 523.141,A -85,B 0,C 180,E1 22862.383,E2 22862.383} C_VEL
LIN {X 0,Y 480.888,Z 523.14,A -85,B 0,C 180,E1 22858.689,E2 22858.689} C_VEL
LIN {X 0,Y 480.871,Z 523.137,A -85,B 0,C 180,E1 22855.109,E2 22855.109} C_VEL
LIN {X 0,Y 480.874,Z 523.135,A -85,B 0,C 180,E1 22851.51,E2 22851.51} C_VEL
LIN {X 0,Y 480.89,Z 523.122,A -85,B 0,C 180,E1 22847.878,E2 22847.878} C_VEL
LIN {X 0,Y 480.877,Z 523.135,A -85,B 0,C 180,E1 22844.302,E2 22844.302} C_VEL
LIN {X 0,Y 480.853,Z 523.137,A -85,B 0,C 180,E1 22840.694,E2 22840.694} C_VEL
LIN {X 0,Y 480.878,Z 523.116,A -85,B 0,C 180,E1 22837.119,E2 22837.119} C_VEL
LIN {X 0,Y 480.882,Z 523.144,A -85,B 0,C 180,E1 22833.58,E2 22833.58} C_VEL
LIN {X 0,Y 480.836,Z 523.12,A -85,B 0,C 180,E1 22830.126,E2 22830.126} C_VEL
LIN {X 0,Y 480.861,Z 523.134,A -85,B 0,C 180,E1 22826.563,E2 22826.563} C_VEL
LIN {X 0,Y 480.873,Z 523.149,A -85,B 0,C 180,E1 22823.065,E2 22823.065} C_VEL
LIN {X 0,Y 480.85,Z 523.298,A -85,B 0,C 180,E1 22819.906,E2 22819.906} C_VEL
LIN {X 0,Y 482.011,Z 526.442,A -85,B 0,C 180,E1 22819.669,E2 22819.669} C_VEL
LIN {X 0,Y 484.677,Z 529.028,A -85,B 0,C 180,E1 22819.238,E2 22819.238} C_VEL
LIN {X 0,Y 487.533,Z 533.4,A -85,B 0,C 180,E1 22818.75,E2 22818.75} C_VEL
LIN {X 0,Y 489.227,Z 535.532,A -85,B 0,C 180,E1 22818.475,E2 22818.475} C_VEL
LIN {X 0,Y 497.231,Z 546.481,A -85,B 0,C 180,E1 22817.204,E2 22817.204} C_VEL
LIN {X 0,Y 507.134,Z 560.475,A -85,B 0,C 180,E1 22815.716,E2 22815.716} C_VEL
LIN {X 0,Y 510.576,Z 565.756,A -85,B 0,C 180,E1 22815.213,E2 22815.213} C_VEL
LIN {X 0,Y 508.877,Z 643.162,A -85,B 0,C 180,E1 22813.896,E2 22813.896} C_VEL
LIN {X 0,Y 507.992,Z 650.865,A -85,B 0,C 180,E1 22813.844,E2 22813.844} C_VEL
LIN {X 0,Y 502.993,Z 671.482,A -85,B 0,C 180,E1 22813.995,E2 22813.995} C_VEL
LIN {X 0,Y 502.316,Z 678.089,A -85,B 0,C 180,E1 22813.942,E2 22813.942} C_VEL
LIN {X 0,Y 498.121,Z 861.682,A -85,B 0,C 180,E1 22810.834,E2 22810.834} C_VEL
LIN {X 0,Y 496.932,Z 885.354,A -85,B 0,C 180,E1 22810.253,E2 22810.253} C_VEL
LIN {X 0,Y 495.579,Z 905.322,A -85,B 0,C 180,E1 22809.582,E2 22809.582} C_VEL
LIN {X 0,Y 493.632,Z 928.135,A -85,B 0,C 180,E1 22808.599,E2 22808.599} C_VEL
LIN {X 0,Y 491.632,Z 948.397,A -85,B 0,C 180,E1 22807.518,E2 22807.518} C_VEL
LIN {X 0,Y 489.35,Z 968.919,A -85,B 0,C 180,E1 22806.188,E2 22806.188} C_VEL
LIN {X 0,Y 487.068,Z 988.105,A -85,B 0,C 180,E1 22804.727,E2 22804.727} C_VEL
LIN {X 0,Y 484.617,Z 1007.483,A -85,B 0,C 180,E1 22803.004,E2 22803.004} C_VEL
LIN {X 0,Y 482.329,Z 1025.896,A -85,B 0,C 180,E1 22801.114,E2 22801.114} C_VEL
LIN {X 0,Y 480.15,Z 1042.716,A -85,B 0,C 180,E1 22799.103,E2 22799.103} C_VEL
LIN {X 0,Y 478.069,Z 1059.89,A -85,B 0,C 180,E1 22796.741,E2 22796.741} C_VEL
LIN {X 0,Y 476.384,Z 1074.47,A -85,B 0,C 180,E1 22794.424,E2 22794.424} C_VEL
LIN {X 0,Y 474.914,Z 1088.226,A -85,B 0,C 180,E1 22791.879,E2 22791.879} C_VEL
LIN {X 0,Y 473.84,Z 1100.069,A -85,B 0,C 180,E1 22789.347,E2 22789.347} C_VEL
LIN {X 0,Y 473.024,Z 1110.443,A -85,B 0,C 180,E1 22786.707,E2 22786.707} C_VEL
LIN {X 0,Y 472.47,Z 1119.507,A -85,B 0,C 180,E1 22783.961,E2 22783.961} C_VEL
LIN {X 0,Y 472.176,Z 1126.147,A -85,B 0,C 180,E1 22781.482,E2 22781.482} C_VEL
LIN {X 0,Y 472.014,Z 1131.939,A -85,B 0,C 180,E1 22778.773,E2 22778.773} C_VEL
LIN {X 0,Y 471.923,Z 1135.899,A -85,B 0,C 180,E1 22776.203,E2 22776.203} C_VEL
LIN {X 0,Y 471.895,Z 1138.687,A -85,B 0,C 180,E1 22773.523,E2 22773.523} C_VEL
LIN {X 0,Y 471.896,Z 1139.818,A -85,B 0,C 180,E1 22770.972,E2 22770.972} C_VEL
LIN {X 0,Y 471.907,Z 1139.722,A -85,B 0,C 180,E1 22768.422,E2 22768.422} C_VEL
LIN {X 0,Y 471.911,Z 1137.998,A -85,B 0,C 180,E1 22765.626,E2 22765.626} C_VEL
LIN {X 0,Y 471.93,Z 1135.22,A -85,B 0,C 180,E1 22763.186,E2 22763.186} C_VEL
LIN {X 0,Y 472.027,Z 1130.43,A -85,B 0,C 180,E1 22760.367,E2 22760.367} C_VEL
LIN {X 0,Y 472.23,Z 1124.854,A -85,B 0,C 180,E1 22757.9,E2 22757.9} C_VEL
LIN {X 0,Y 472.638,Z 1116.701,A -85,B 0,C 180,E1 22755.043,E2 22755.043} C_VEL
LIN {X 0,Y 473.214,Z 1108.012,A -85,B 0,C 180,E1 22752.541,E2 22752.541} C_VEL
LIN {X 0,Y 474.154,Z 1096.493,A -85,B 0,C 180,E1 22749.768,E2 22749.768} C_VEL
LIN {X 0,Y 475.361,Z 1084.188,A -85,B 0,C 180,E1 22747.231,E2 22747.231} C_VEL
LIN {X 0,Y 476.829,Z 1070.375,A -85,B 0,C 180,E1 22744.807,E2 22744.807} C_VEL
LIN {X 0,Y 478.763,Z 1053.962,A -85,B 0,C 180,E1 22742.312,E2 22742.312} C_VEL
LIN {X 0,Y 480.797,Z 1037.88,A -85,B 0,C 180,E1 22740.197,E2 22740.197} C_VEL
LIN {X 0,Y 483.058,Z 1019.779,A -85,B 0,C 180,E1 22738.142,E2 22738.142} C_VEL
LIN {X 0,Y 485.459,Z 1001.22,A -85,B 0,C 180,E1 22736.314,E2 22736.314} C_VEL
LIN {X 0,Y 487.992,Z 980.297,A -85,B 0,C 180,E1 22734.56,E2 22734.56} C_VEL
LIN {X 0,Y 490.404,Z 959.726,A -85,B 0,C 180,E1 22733.099,E2 22733.099} C_VEL
LIN {X 0,Y 492.433,Z 940.793,A -85,B 0,C 180,E1 22731.965,E2 22731.965} C_VEL
LIN {X 0,Y 494.517,Z 918.171,A -85,B 0,C 180,E1 22730.851,E2 22730.851} C_VEL
LIN {X 0,Y 496.188,Z 896.743,A -85,B 0,C 180,E1 22730.012,E2 22730.012} C_VEL
LIN {X 0,Y 497.541,Z 874.351,A -85,B 0,C 180,E1 22729.36,E2 22729.36} C_VEL
LIN {X 0,Y 498.495,Z 851.304,A -85,B 0,C 180,E1 22728.882,E2 22728.882} C_VEL
LIN {X 0,Y 503.06,Z 647.241,A -85,B 0,C 180,E1 22725.446,E2 22725.446} C_VEL
LIN {X 0,Y 504.786,Z 569.078,A -85,B 0,C 180,E1 22724.09,E2 22724.09} C_VEL
LIN {X 0,Y 491.453,Z 550.009,A -85,B 0,C 180,E1 22722.04,E2 22722.04} C_VEL
LIN {X 0,Y 483.6,Z 539.529,A -85,B 0,C 180,E1 22720.755,E2 22720.755} C_VEL
LIN {X 0,Y 480.449,Z 535.22,A -85,B 0,C 180,E1 22720.215,E2 22720.215} C_VEL
LIN {X 0,Y 477.594,Z 531.605,A -85,B 0,C 180,E1 22719.721,E2 22719.721} C_VEL
LIN {X 0,Y 476.643,Z 529.921,A -85,B 0,C 180,E1 22719.543,E2 22719.543} C_VEL
LIN {X 0,Y 473.98,Z 527.183,A -85,B 0,C 180,E1 22719.083,E2 22719.083} C_VEL
LIN {X 0,Y 472.906,Z 524.11,A -85,B 0,C 180,E1 22718.841,E2 22718.841} C_VEL
LIN {X 0,Y 472.919,Z 524.112,A -85,B 0,C 180,E1 22715.401,E2 22715.401} C_VEL
LIN {X 0,Y 472.894,Z 524.142,A -85,B 0,C 180,E1 22711.91,E2 22711.91} C_VEL
LIN {X 0,Y 472.928,Z 524.11,A -85,B 0,C 180,E1 22708.405,E2 22708.405} C_VEL
LIN {X 0,Y 472.936,Z 524.113,A -85,B 0,C 180,E1 22704.88,E2 22704.88} C_VEL
LIN {X 0,Y 472.908,Z 524.132,A -85,B 0,C 180,E1 22701.325,E2 22701.325} C_VEL
LIN {X 0,Y 472.925,Z 524.101,A -85,B 0,C 180,E1 22697.725,E2 22697.725} C_VEL
LIN {X 0,Y 472.954,Z 524.134,A -85,B 0,C 180,E1 22694.196,E2 22694.196} C_VEL
LIN {X 0,Y 472.931,Z 524.135,A -85,B 0,C 180,E1 22690.551,E2 22690.551} C_VEL
LIN {X 0,Y 472.927,Z 524.135,A -85,B 0,C 180,E1 22686.922,E2 22686.922} C_VEL
LIN {X 0,Y 472.95,Z 524.134,A -85,B 0,C 180,E1 22683.273,E2 22683.273} C_VEL
LIN {X 0,Y 472.951,Z 524.137,A -85,B 0,C 180,E1 22679.637,E2 22679.637} C_VEL
LIN {X 0,Y 472.94,Z 524.134,A -85,B 0,C 180,E1 22676,E2 22676} C_VEL
LIN {X 0,Y 472.945,Z 524.132,A -85,B 0,C 180,E1 22672.346,E2 22672.346} C_VEL
LIN {X 0,Y 472.934,Z 524.095,A -85,B 0,C 180,E1 22668.785,E2 22668.785} C_VEL
LIN {X 0,Y 472.942,Z 524.135,A -85,B 0,C 180,E1 22665.051,E2 22665.051} C_VEL
LIN {X 0,Y 472.946,Z 524.103,A -85,B 0,C 180,E1 22661.384,E2 22661.384} C_VEL
LIN {X 0,Y 472.956,Z 524.12,A -85,B 0,C 180,E1 22657.765,E2 22657.765} C_VEL
LIN {X 0,Y 472.924,Z 524.136,A -85,B 0,C 180,E1 22654.182,E2 22654.182} C_VEL
LIN {X 0,Y 472.936,Z 524.106,A -85,B 0,C 180,E1 22650.579,E2 22650.579} C_VEL
LIN {X 0,Y 472.953,Z 524.112,A -85,B 0,C 180,E1 22646.946,E2 22646.946} C_VEL
LIN {X 0,Y 472.917,Z 524.136,A -85,B 0,C 180,E1 22643.401,E2 22643.401} C_VEL
LIN {X 0,Y 472.98,Z 524.344,A -85,B 0,C 180,E1 22642.858,E2 22642.858} C_VEL
LIN {X 0,Y 474.251,Z 527.609,A -85,B 0,C 180,E1 22642.309,E2 22642.309} C_VEL
LIN {X 0,Y 475.38,Z 529.325,A -85,B 0,C 180,E1 22641.957,E2 22641.957} C_VEL
LIN {X 0,Y 477.464,Z 533.275,A -85,B 0,C 180,E1 22641.235,E2 22641.235} C_VEL
LIN {X 0,Y 480.851,Z 540.166,A -85,B 0,C 180,E1 22640.098,E2 22640.098} C_VEL
LIN {X 0,Y 487.683,Z 549.964,A -85,B 0,C 180,E1 22638.941,E2 22638.941} C_VEL
LIN {X 0,Y 498.531,Z 566.253,A -85,B 0,C 180,E1 22637.204,E2 22637.204} C_VEL
LIN {X 0,Y 505.132,Z 576.962,A -85,B 0,C 180,E1 22636.193,E2 22636.193} C_VEL
LIN {X 0,Y 500.806,Z 766.935,A -85,B 0,C 180,E1 22632.96,E2 22632.96} C_VEL
LIN {X 0,Y 497.959,Z 891.654,A -85,B 0,C 180,E1 22630.857,E2 22630.857} C_VEL
LIN {X 0,Y 496.742,Z 914.601,A -85,B 0,C 180,E1 22630.286,E2 22630.286} C_VEL
LIN {X 0,Y 495.321,Z 935.594,A -85,B 0,C 180,E1 22629.581,E2 22629.581} C_VEL
LIN {X 0,Y 493.419,Z 957.84,A -85,B 0,C 180,E1 22628.618,E2 22628.618} C_VEL
LIN {X 0,Y 491.362,Z 979.338,A -85,B 0,C 180,E1 22627.476,E2 22627.476} C_VEL
LIN {X 0,Y 489.161,Z 999.652,A -85,B 0,C 180,E1 22626.159,E2 22626.159} C_VEL
LIN {X 0,Y 486.917,Z 1019.424,A -85,B 0,C 180,E1 22624.667,E2 22624.667} C_VEL
LIN {X 0,Y 484.48,Z 1038.589,A -85,B 0,C 180,E1 22622.943,E2 22622.943} C_VEL
LIN {X 0,Y 482.083,Z 1057.672,A -85,B 0,C 180,E1 22620.955,E2 22620.955} C_VEL
LIN {X 0,Y 479.979,Z 1074.153,A -85,B 0,C 180,E1 22618.966,E2 22618.966} C_VEL
LIN {X 0,Y 478.015,Z 1090.292,A -85,B 0,C 180,E1 22616.725,E2 22616.725} C_VEL
LIN {X 0,Y 476.312,Z 1105.174,A -85,B 0,C 180,E1 22614.352,E2 22614.352} C_VEL
LIN {X 0,Y 474.892,Z 1118.446,A -85,B 0,C 180,E1 22611.88,E2 22611.88} C_VEL
LIN {X 0,Y 473.82,Z 1130.25,A -85,B 0,C 180,E1 22609.348,E2 22609.348} C_VEL
LIN {X 0,Y 473.028,Z 1140.408,A -85,B 0,C 180,E1 22606.761,E2 22606.761} C_VEL
LIN {X 0,Y 472.461,Z 1149.638,A -85,B 0,C 180,E1 22603.96,E2 22603.96} C_VEL
LIN {X 0,Y 472.17,Z 1156.259,A -85,B 0,C 180,E1 22601.481,E2 22601.481} C_VEL
LIN {X 0,Y 472.004,Z 1162.222,A -85,B 0,C 180,E1 22598.65,E2 22598.65} C_VEL
LIN {X 0,Y 471.918,Z 1166.119,A -85,B 0,C 180,E1 22596.081,E2 22596.081} C_VEL
LIN {X 0,Y 471.886,Z 1168.85,A -85,B 0,C 180,E1 22593.279,E2 22593.279} C_VEL
LIN {X 0,Y 471.887,Z 1169.849,A -85,B 0,C 180,E1 22590.85,E2 22590.85} C_VEL
LIN {X 0,Y 471.905,Z 1169.658,A -85,B 0,C 180,E1 22588.178,E2 22588.178} C_VEL
LIN {X 0,Y 471.91,Z 1167.841,A -85,B 0,C 180,E1 22585.503,E2 22585.503} C_VEL
LIN {X 0,Y 471.928,Z 1164.68,A -85,B 0,C 180,E1 22582.819,E2 22582.819} C_VEL
LIN {X 0,Y 472.031,Z 1160.081,A -85,B 0,C 180,E1 22580.243,E2 22580.243} C_VEL
LIN {X 0,Y 472.244,Z 1154.436,A -85,B 0,C 180,E1 22577.776,E2 22577.776} C_VEL
LIN {X 0,Y 472.667,Z 1146.149,A -85,B 0,C 180,E1 22574.918,E2 22574.918} C_VEL
LIN {X 0,Y 473.301,Z 1136.921,A -85,B 0,C 180,E1 22572.289,E2 22572.289} C_VEL
LIN {X 0,Y 474.22,Z 1125.72,A -85,B 0,C 180,E1 22569.641,E2 22569.641} C_VEL
LIN {X 0,Y 475.457,Z 1113.142,A -85,B 0,C 180,E1 22567.085,E2 22567.085} C_VEL
LIN {X 0,Y 476.952,Z 1099.339,A -85,B 0,C 180,E1 22564.681,E2 22564.681} C_VEL
LIN {X 0,Y 478.852,Z 1083.178,A -85,B 0,C 180,E1 22562.248,E2 22562.248} C_VEL
LIN {X 0,Y 480.981,Z 1066.526,A -85,B 0,C 180,E1 22560.072,E2 22560.072} C_VEL
LIN {X 0,Y 483.196,Z 1048.709,A -85,B 0,C 180,E1 22558.075,E2 22558.075} C_VEL
LIN {X 0,Y 485.628,Z 1029.707,A -85,B 0,C 180,E1 22556.227,E2 22556.227} C_VEL
LIN {X 0,Y 487.733,Z 1012.067,A -85,B 0,C 180,E1 22554.754,E2 22554.754} C_VEL
LIN {X 0,Y 490.066,Z 991.565,A -85,B 0,C 180,E1 22553.287,E2 22553.287} C_VEL
LIN {X 0,Y 492.154,Z 971.356,A -85,B 0,C 180,E1 22552.08,E2 22552.08} C_VEL
LIN {X 0,Y 494.206,Z 949.124,A -85,B 0,C 180,E1 22550.976,E2 22550.976} C_VEL
LIN {X 0,Y 495.839,Z 927.921,A -85,B 0,C 180,E1 22550.138,E2 22550.138} C_VEL
LIN {X 0,Y 497.363,Z 903.884,A -85,B 0,C 180,E1 22549.423,E2 22549.423} C_VEL
LIN {X 0,Y 498.3,Z 882.002,A -85,B 0,C 180,E1 22548.963,E2 22548.963} C_VEL
LIN {X 0,Y 502.69,Z 681.501,A -85,B 0,C 180,E1 22545.594,E2 22545.594} C_VEL
LIN {X 0,Y 505.026,Z 576.446,A -85,B 0,C 180,E1 22543.784,E2 22543.784} C_VEL
LIN {X 0,Y 491.557,Z 555.589,A -85,B 0,C 180,E1 22541.692,E2 22541.692} C_VEL
LIN {X 0,Y 482.126,Z 541.906,A -85,B 0,C 180,E1 22540.124,E2 22540.124} C_VEL
LIN {X 0,Y 480.179,Z 538.916,A -85,B 0,C 180,E1 22539.736,E2 22539.736} C_VEL
LIN {X 0,Y 477.034,Z 532.747,A -85,B 0,C 180,E1 22538.653,E2 22538.653} C_VEL
LIN {X 0,Y 474.657,Z 528.191,A -85,B 0,C 180,E1 22537.82,E2 22537.82} C_VEL
LIN {X 0,Y 473.038,Z 524.668,A -85,B 0,C 180,E1 22537.194,E2 22537.194} C_VEL
LIN {X 0,Y 472.946,Z 524.133,A -85,B 0,C 180,E1 22537.05,E2 22537.05} C_VEL
LIN {X 0,Y 472.946,Z 524.109,A -85,B 0,C 180,E1 22533.376,E2 22533.376} C_VEL
LIN {X 0,Y 472.915,Z 524.107,A -85,B 0,C 180,E1 22529.791,E2 22529.791} C_VEL
LIN {X 0,Y 472.929,Z 524.133,A -85,B 0,C 180,E1 22526.088,E2 22526.088} C_VEL
LIN {X 0,Y 472.948,Z 524.107,A -85,B 0,C 180,E1 22522.498,E2 22522.498} C_VEL
LIN {X 0,Y 472.943,Z 524.108,A -85,B 0,C 180,E1 22518.872,E2 22518.872} C_VEL
LIN {X 0,Y 472.931,Z 524.129,A -85,B 0,C 180,E1 22515.198,E2 22515.198} C_VEL
LIN {X 0,Y 472.944,Z 524.1,A -85,B 0,C 180,E1 22511.586,E2 22511.586} C_VEL
LIN {X 0,Y 472.941,Z 524.136,A -85,B 0,C 180,E1 22507.898,E2 22507.898} C_VEL
LIN {X 0,Y 472.947,Z 524.135,A -85,B 0,C 180,E1 22504.243,E2 22504.243} C_VEL
LIN {X 0,Y 472.944,Z 524.133,A -85,B 0,C 180,E1 22500.605,E2 22500.605} C_VEL
LIN {X 0,Y 472.944,Z 524.133,A -85,B 0,C 180,E1 22496.97,E2 22496.97} C_VEL
LIN {X 0,Y 472.929,Z 524.138,A -85,B 0,C 180,E1 22493.322,E2 22493.322} C_VEL
LIN {X 0,Y 472.944,Z 524.095,A -85,B 0,C 180,E1 22489.771,E2 22489.771} C_VEL
LIN {X 0,Y 472.955,Z 524.133,A -85,B 0,C 180,E1 22486.054,E2 22486.054} C_VEL
LIN {X 0,Y 472.917,Z 524.095,A -85,B 0,C 180,E1 22482.465,E2 22482.465} C_VEL
LIN {X 0,Y 472.917,Z 524.136,A -85,B 0,C 180,E1 22478.805,E2 22478.805} C_VEL
LIN {X 0,Y 472.949,Z 524.101,A -85,B 0,C 180,E1 22475.254,E2 22475.254} C_VEL
LIN {X 0,Y 472.919,Z 524.12,A -85,B 0,C 180,E1 22471.732,E2 22471.732} C_VEL
LIN {X 0,Y 472.902,Z 524.141,A -85,B 0,C 180,E1 22468.207,E2 22468.207} C_VEL
LIN {X 0,Y 472.938,Z 524.107,A -85,B 0,C 180,E1 22464.693,E2 22464.693} C_VEL
LIN {X 0,Y 472.902,Z 524.114,A -85,B 0,C 180,E1 22461.256,E2 22461.256} C_VEL
LIN {X 0,Y 472.938,Z 524.247,A -85,B 0,C 180,E1 22461.048,E2 22461.048} C_VEL
LIN {X 0,Y 474.132,Z 527.407,A -85,B 0,C 180,E1 22460.793,E2 22460.793} C_VEL
LIN {X 0,Y 477.073,Z 530.535,A -85,B 0,C 180,E1 22460.285,E2 22460.285} C_VEL
LIN {X 0,Y 479.655,Z 534.45,A -85,B 0,C 180,E1 22459.822,E2 22459.822} C_VEL
LIN {X 0,Y 481.475,Z 536.484,A -85,B 0,C 180,E1 22459.517,E2 22459.517} C_VEL
LIN {X 0,Y 493.016,Z 552.266,A -85,B 0,C 180,E1 22457.618,E2 22457.618} C_VEL
LIN {X 0,Y 504.885,Z 569.178,A -85,B 0,C 180,E1 22455.806,E2 22455.806} C_VEL
LIN {X 0,Y 502.316,Z 678.089,A -85,B 0,C 180,E1 22453.942,E2 22453.942} C_VEL
LIN {X 0,Y 501.438,Z 685.79,A -85,B 0,C 180,E1 22453.888,E2 22453.888} C_VEL
LIN {X 0,Y 496.438,Z 706.407,A -85,B 0,C 180,E1 22454.042,E2 22454.042} C_VEL
LIN {X 0,Y 495.754,Z 713.015,A -85,B 0,C 180,E1 22453.988,E2 22453.988} C_VEL
LIN {X 0,Y 492.052,Z 863.375,A -85,B 0,C 180,E1 22451.417,E2 22451.417} C_VEL
LIN {X 0,Y 490.803,Z 886.251,A -85,B 0,C 180,E1 22450.84,E2 22450.84} C_VEL
LIN {X 0,Y 489.341,Z 906.635,A -85,B 0,C 180,E1 22450.145,E2 22450.145} C_VEL
LIN {X 0,Y 487.357,Z 928.454,A -85,B 0,C 180,E1 22449.19,E2 22449.19} C_VEL
LIN {X 0,Y 485.366,Z 947.471,A -85,B 0,C 180,E1 22448.171,E2 22448.171} C_VEL
LIN {X 0,Y 482.804,Z 969.181,A -85,B 0,C 180,E1 22446.763,E2 22446.763} C_VEL
LIN {X 0,Y 480.382,Z 988.342,A -85,B 0,C 180,E1 22445.289,E2 22445.289} C_VEL
LIN {X 0,Y 477.713,Z 1007.577,A -85,B 0,C 180,E1 22443.543,E2 22443.543} C_VEL
LIN {X 0,Y 475.024,Z 1027.311,A -85,B 0,C 180,E1 22441.467,E2 22441.467} C_VEL
LIN {X 0,Y 472.75,Z 1043.804,A -85,B 0,C 180,E1 22439.455,E2 22439.455} C_VEL
LIN {X 0,Y 470.509,Z 1060.853,A -85,B 0,C 180,E1 22437.05,E2 22437.05} C_VEL
LIN {X 0,Y 468.691,Z 1075.558,A -85,B 0,C 180,E1 22434.662,E2 22434.662} C_VEL
LIN {X 0,Y 467.144,Z 1088.863,A -85,B 0,C 180,E1 22432.13,E2 22432.13} C_VEL
LIN {X 0,Y 465.934,Z 1101.116,A -85,B 0,C 180,E1 22429.428,E2 22429.428} C_VEL
LIN {X 0,Y 465.11,Z 1110.903,A -85,B 0,C 180,E1 22426.871,E2 22426.871} C_VEL
LIN {X 0,Y 464.489,Z 1120.219,A -85,B 0,C 180,E1 22423.951,E2 22423.951} C_VEL
LIN {X 0,Y 464.173,Z 1127.058,A -85,B 0,C 180,E1 22421.305,E2 22421.305} C_VEL
LIN {X 0,Y 463.996,Z 1132.767,A -85,B 0,C 180,E1 22418.426,E2 22418.426} C_VEL
LIN {X 0,Y 463.908,Z 1136.538,A -85,B 0,C 180,E1 22415.814,E2 22415.814} C_VEL
LIN {X 0,Y 463.885,Z 1138.96,A -85,B 0,C 180,E1 22413.089,E2 22413.089} C_VEL
LIN {X 0,Y 463.887,Z 1139.886,A -85,B 0,C 180,E1 22410.618,E2 22410.618} C_VEL
LIN {X 0,Y 463.913,Z 1139.485,A -85,B 0,C 180,E1 22407.777,E2 22407.777} C_VEL
LIN {X 0,Y 463.91,Z 1137.656,A -85,B 0,C 180,E1 22405.178,E2 22405.178} C_VEL
LIN {X 0,Y 463.955,Z 1134.156,A -85,B 0,C 180,E1 22402.322,E2 22402.322} C_VEL
LIN {X 0,Y 464.06,Z 1129.665,A -85,B 0,C 180,E1 22399.824,E2 22399.824} C_VEL
LIN {X 0,Y 464.32,Z 1123.632,A -85,B 0,C 180,E1 22397.186,E2 22397.186} C_VEL
LIN {X 0,Y 464.799,Z 1115.482,A -85,B 0,C 180,E1 22394.402,E2 22394.402} C_VEL
LIN {X 0,Y 465.561,Z 1105.59,A -85,B 0,C 180,E1 22391.597,E2 22391.597} C_VEL
LIN {X 0,Y 466.552,Z 1094.767,A -85,B 0,C 180,E1 22389.029,E2 22389.029} C_VEL
LIN {X 0,Y 467.988,Z 1081.383,A -85,B 0,C 180,E1 22386.318,E2 22386.318} C_VEL
LIN {X 0,Y 469.626,Z 1067.886,A -85,B 0,C 180,E1 22383.957,E2 22383.957} C_VEL
LIN {X 0,Y 471.598,Z 1052.42,A -85,B 0,C 180,E1 22381.626,E2 22381.626} C_VEL
LIN {X 0,Y 473.894,Z 1035.58,A -85,B 0,C 180,E1 22379.41,E2 22379.41} C_VEL
LIN {X 0,Y 476.291,Z 1017.944,A -85,B 0,C 180,E1 22377.421,E2 22377.421} C_VEL
LIN {X 0,Y 479.113,Z 997.448,A -85,B 0,C 180,E1 22375.415,E2 22375.415} C_VEL
LIN {X 0,Y 481.705,Z 978.184,A -85,B 0,C 180,E1 22373.806,E2 22373.806} C_VEL
LIN {X 0,Y 484.165,Z 958.027,A -85,B 0,C 180,E1 22372.393,E2 22372.393} C_VEL
LIN {X 0,Y 486.471,Z 937.599,A -85,B 0,C 180,E1 22371.18,E2 22371.18} C_VEL
LIN {X 0,Y 488.531,Z 915.613,A -85,B 0,C 180,E1 22370.13,E2 22370.13} C_VEL
LIN {X 0,Y 490.392,Z 892.71,A -85,B 0,C 180,E1 22369.269,E2 22369.269} C_VEL
LIN {X 0,Y 491.603,Z 872.677,A -85,B 0,C 180,E1 22368.706,E2 22368.706} C_VEL
LIN {X 0,Y 492.581,Z 847.624,A -85,B 0,C 180,E1 22368.204,E2 22368.204} C_VEL
LIN {X 0,Y 497.515,Z 642.534,A -85,B 0,C 180,E1 22364.715,E2 22364.715} C_VEL
LIN {X 0,Y 499.121,Z 572.94,A -85,B 0,C 180,E1 22363.489,E2 22363.489} C_VEL
LIN {X 0,Y 487.477,Z 556.108,A -85,B 0,C 180,E1 22361.648,E2 22361.648} C_VEL
LIN {X 0,Y 476.656,Z 541.545,A -85,B 0,C 180,E1 22359.815,E2 22359.815} C_VEL
LIN {X 0,Y 473.434,Z 537.129,A -85,B 0,C 180,E1 22359.237,E2 22359.237} C_VEL
LIN {X 0,Y 469.804,Z 532.613,A -85,B 0,C 180,E1 22358.578,E2 22358.578} C_VEL
LIN {X 0,Y 468.726,Z 530.953,A -85,B 0,C 180,E1 22358.371,E2 22358.371} C_VEL
LIN {X 0,Y 466.132,Z 528.406,A -85,B 0,C 180,E1 22357.9,E2 22357.9} C_VEL
LIN {X 0,Y 464.989,Z 525.276,A -85,B 0,C 180,E1 22357.639,E2 22357.639} C_VEL
LIN {X 0,Y 464.948,Z 525.098,A -85,B 0,C 180,E1 22354.113,E2 22354.113} C_VEL
LIN {X 0,Y 465.001,Z 525.103,A -85,B 0,C 180,E1 22350.638,E2 22350.638} C_VEL
LIN {X 0,Y 464.988,Z 525.122,A -85,B 0,C 180,E1 22347.099,E2 22347.099} C_VEL
LIN {X 0,Y 464.961,Z 525.088,A -85,B 0,C 180,E1 22343.577,E2 22343.577} C_VEL
LIN {X 0,Y 465,Z 525.123,A -85,B 0,C 180,E1 22339.992,E2 22339.992} C_VEL
LIN {X 0,Y 465.009,Z 525.084,A -85,B 0,C 180,E1 22336.36,E2 22336.36} C_VEL
LIN {X 0,Y 464.984,Z 525.125,A -85,B 0,C 180,E1 22332.796,E2 22332.796} C_VEL
LIN {X 0,Y 464.987,Z 525.122,A -85,B 0,C 180,E1 22329.031,E2 22329.031} C_VEL
LIN {X 0,Y 465.01,Z 525.115,A -85,B 0,C 180,E1 22325.415,E2 22325.415} C_VEL
LIN {X 0,Y 465.01,Z 525.115,A -85,B 0,C 180,E1 22321.725,E2 22321.725} C_VEL
LIN {X 0,Y 464.997,Z 525.12,A -85,B 0,C 180,E1 22318.152,E2 22318.152} C_VEL
LIN {X 0,Y 465.004,Z 525.118,A -85,B 0,C 180,E1 22314.448,E2 22314.448} C_VEL
LIN {X 0,Y 465.001,Z 525.113,A -85,B 0,C 180,E1 22310.845,E2 22310.845} C_VEL
LIN {X 0,Y 464.999,Z 525.103,A -85,B 0,C 180,E1 22307.078,E2 22307.078} C_VEL
LIN {X 0,Y 465.005,Z 525.097,A -85,B 0,C 180,E1 22303.512,E2 22303.512} C_VEL
LIN {X 0,Y 465.012,Z 525.122,A -85,B 0,C 180,E1 22299.747,E2 22299.747} C_VEL
LIN {X 0,Y 464.984,Z 525.091,A -85,B 0,C 180,E1 22296.156,E2 22296.156} C_VEL
LIN {X 0,Y 464.988,Z 525.116,A -85,B 0,C 180,E1 22292.464,E2 22292.464} C_VEL
LIN {X 0,Y 465.016,Z 525.119,A -85,B 0,C 180,E1 22288.844,E2 22288.844} C_VEL
LIN {X 0,Y 464.996,Z 525.097,A -85,B 0,C 180,E1 22285.225,E2 22285.225} C_VEL
LIN {X 0,Y 465,Z 525.294,A -85,B 0,C 180,E1 22284.012,E2 22284.012} C_VEL
LIN {X 0,Y 466.333,Z 528.681,A -85,B 0,C 180,E1 22283.413,E2 22283.413} C_VEL
LIN {X 0,Y 467.507,Z 530.169,A -85,B 0,C 180,E1 22283.061,E2 22283.061} C_VEL
LIN {X 0,Y 469.459,Z 534.153,A -85,B 0,C 180,E1 22282.32,E2 22282.32} C_VEL
LIN {X 0,Y 472.46,Z 539.717,A -85,B 0,C 180,E1 22281.331,E2 22281.331} C_VEL
LIN {X 0,Y 483.388,Z 555.532,A -85,B 0,C 180,E1 22279.4,E2 22279.4} C_VEL
LIN {X 0,Y 494.197,Z 571.897,A -85,B 0,C 180,E1 22277.626,E2 22277.626} C_VEL
LIN {X 0,Y 499.483,Z 580.655,A -85,B 0,C 180,E1 22276.791,E2 22276.791} C_VEL
LIN {X 0,Y 494.817,Z 771.925,A -85,B 0,C 180,E1 22273.506,E2 22273.506} C_VEL
LIN {X 0,Y 491.897,Z 891.352,A -85,B 0,C 180,E1 22271.47,E2 22271.47} C_VEL
LIN {X 0,Y 490.585,Z 914.483,A -85,B 0,C 180,E1 22270.891,E2 22270.891} C_VEL
LIN {X 0,Y 489.024,Z 936.167,A -85,B 0,C 180,E1 22270.155,E2 22270.155} C_VEL
LIN {X 0,Y 487.069,Z 957.534,A -85,B 0,C 180,E1 22269.217,E2 22269.217} C_VEL
LIN {X 0,Y 484.979,Z 977.891,A -85,B 0,C 180,E1 22268.131,E2 22268.131} C_VEL
LIN {X 0,Y 482.573,Z 998.724,A -85,B 0,C 180,E1 22266.783,E2 22266.783} C_VEL
LIN {X 0,Y 480.112,Z 1019.14,A -85,B 0,C 180,E1 22265.23,E2 22265.23} C_VEL
LIN {X 0,Y 477.537,Z 1038.534,A -85,B 0,C 180,E1 22263.484,E2 22263.484} C_VEL
LIN {X 0,Y 475.217,Z 1056.006,A -85,B 0,C 180,E1 22261.665,E2 22261.665} C_VEL
LIN {X 0,Y 472.845,Z 1073.122,A -85,B 0,C 180,E1 22259.587,E2 22259.587} C_VEL
LIN {X 0,Y 470.584,Z 1090.29,A -85,B 0,C 180,E1 22257.182,E2 22257.182} C_VEL
LIN {X 0,Y 468.78,Z 1104.734,A -85,B 0,C 180,E1 22254.846,E2 22254.846} C_VEL
LIN {X 0,Y 467.263,Z 1117.809,A -85,B 0,C 180,E1 22252.389,E2 22252.389} C_VEL
LIN {X 0,Y 466.08,Z 1129.725,A -85,B 0,C 180,E1 22249.813,E2 22249.813} C_VEL
LIN {X 0,Y 465.17,Z 1140.146,A -85,B 0,C 180,E1 22247.126,E2 22247.126} C_VEL
LIN {X 0,Y 464.55,Z 1149.283,A -85,B 0,C 180,E1 22244.33,E2 22244.33} C_VEL
LIN {X 0,Y 464.217,Z 1155.956,A -85,B 0,C 180,E1 22241.807,E2 22241.807} C_VEL
LIN {X 0,Y 464.029,Z 1161.809,A -85,B 0,C 180,E1 22239.05,E2 22239.05} C_VEL
LIN {X 0,Y 463.932,Z 1165.96,A -85,B 0,C 180,E1 22236.31,E2 22236.31} C_VEL
LIN {X 0,Y 463.896,Z 1168.713,A -85,B 0,C 180,E1 22233.583,E2 22233.583} C_VEL
LIN {X 0,Y 463.892,Z 1169.827,A -85,B 0,C 180,E1 22230.988,E2 22230.988} C_VEL
LIN {X 0,Y 463.905,Z 1169.713,A -85,B 0,C 180,E1 22228.394,E2 22228.394} C_VEL
LIN {X 0,Y 463.911,Z 1167.955,A -85,B 0,C 180,E1 22225.55,E2 22225.55} C_VEL
LIN {X 0,Y 463.928,Z 1165,A -85,B 0,C 180,E1 22222.943,E2 22222.943} C_VEL
LIN {X 0,Y 464.039,Z 1160.335,A -85,B 0,C 180,E1 22220.199,E2 22220.199} C_VEL
LIN {X 0,Y 464.265,Z 1154.741,A -85,B 0,C 180,E1 22217.689,E2 22217.689} C_VEL
LIN {X 0,Y 464.724,Z 1146.552,A -85,B 0,C 180,E1 22214.782,E2 22214.782} C_VEL
LIN {X 0,Y 465.363,Z 1137.85,A -85,B 0,C 180,E1 22212.236,E2 22212.236} C_VEL
LIN {X 0,Y 466.341,Z 1126.865,A -85,B 0,C 180,E1 22209.544,E2 22209.544} C_VEL
LIN {X 0,Y 467.644,Z 1114.618,A -85,B 0,C 180,E1 22206.966,E2 22206.966} C_VEL
LIN {X 0,Y 469.232,Z 1100.878,A -85,B 0,C 180,E1 22204.505,E2 22204.505} C_VEL
LIN {X 0,Y 471.185,Z 1085.609,A -85,B 0,C 180,E1 22202.119,E2 22202.119} C_VEL
LIN {X 0,Y 473.342,Z 1069.57,A -85,B 0,C 180,E1 22199.958,E2 22199.958} C_VEL
LIN {X 0,Y 475.858,Z 1050.999,A -85,B 0,C 180,E1 22197.791,E2 22197.791} C_VEL
LIN {X 0,Y 478.001,Z 1035.141,A -85,B 0,C 180,E1 22196.192,E2 22196.192} C_VEL
LIN {X 0,Y 480.68,Z 1014.216,A -85,B 0,C 180,E1 22194.378,E2 22194.378} C_VEL
LIN {X 0,Y 483.142,Z 994.174,A -85,B 0,C 180,E1 22192.896,E2 22192.896} C_VEL
LIN {X 0,Y 485.464,Z 973.328,A -85,B 0,C 180,E1 22191.613,E2 22191.613} C_VEL
LIN {X 0,Y 487.609,Z 952.35,A -85,B 0,C 180,E1 22190.53,E2 22190.53} C_VEL
LIN {X 0,Y 489.472,Z 929.796,A -85,B 0,C 180,E1 22189.609,E2 22189.609} C_VEL
LIN {X 0,Y 491.096,Z 906.678,A -85,B 0,C 180,E1 22188.886,E2 22188.886} C_VEL
LIN {X 0,Y 492.154,Z 884.492,A -85,B 0,C 180,E1 22188.401,E2 22188.401} C_VEL
LIN {X 0,Y 496.848,Z 685.922,A -85,B 0,C 180,E1 22185.025,E2 22185.025} C_VEL
LIN {X 0,Y 499.339,Z 580.122,A -85,B 0,C 180,E1 22183.181,E2 22183.181} C_VEL
LIN {X 0,Y 487.216,Z 561.166,A -85,B 0,C 180,E1 22181.243,E2 22181.243} C_VEL
LIN {X 0,Y 478.171,Z 547.932,A -85,B 0,C 180,E1 22179.702,E2 22179.702} C_VEL
LIN {X 0,Y 471.833,Z 538.749,A -85,B 0,C 180,E1 22178.536,E2 22178.536} C_VEL
LIN {X 0,Y 467.49,Z 530.144,A -85,B 0,C 180,E1 22176.941,E2 22176.941} C_VEL
LIN {X 0,Y 465.346,Z 526.749,A -85,B 0,C 180,E1 22176.219,E2 22176.219} C_VEL
LIN {X 0,Y 464.976,Z 525.125,A -85,B 0,C 180,E1 22175.947,E2 22175.947} C_VEL
LIN {X 0,Y 464.978,Z 525.126,A -85,B 0,C 180,E1 22172.227,E2 22172.227} C_VEL
LIN {X 0,Y 465.015,Z 525.088,A -85,B 0,C 180,E1 22168.651,E2 22168.651} C_VEL
LIN {X 0,Y 465.005,Z 525.098,A -85,B 0,C 180,E1 22165.061,E2 22165.061} C_VEL
LIN {X 0,Y 464.989,Z 525.118,A -85,B 0,C 180,E1 22161.396,E2 22161.396} C_VEL
LIN {X 0,Y 464.994,Z 525.081,A -85,B 0,C 180,E1 22157.716,E2 22157.716} C_VEL
LIN {X 0,Y 465.01,Z 525.123,A -85,B 0,C 180,E1 22154.062,E2 22154.062} C_VEL
LIN {X 0,Y 465.004,Z 525.083,A -85,B 0,C 180,E1 22150.405,E2 22150.405} C_VEL
LIN {X 0,Y 465.003,Z 525.126,A -85,B 0,C 180,E1 22146.791,E2 22146.791} C_VEL
LIN {X 0,Y 465.008,Z 525.122,A -85,B 0,C 180,E1 22143.081,E2 22143.081} C_VEL
LIN {X 0,Y 464.997,Z 525.12,A -85,B 0,C 180,E1 22139.384,E2 22139.384} C_VEL
LIN {X 0,Y 464.998,Z 525.119,A -85,B 0,C 180,E1 22135.684,E2 22135.684} C_VEL
LIN {X 0,Y 465.011,Z 525.12,A -85,B 0,C 180,E1 22132.09,E2 22132.09} C_VEL
LIN {X 0,Y 465.005,Z 525.089,A -85,B 0,C 180,E1 22128.339,E2 22128.339} C_VEL
LIN {X 0,Y 464.982,Z 525.119,A -85,B 0,C 180,E1 22124.791,E2 22124.791} C_VEL
LIN {X 0,Y 464.989,Z 525.098,A -85,B 0,C 180,E1 22121.109,E2 22121.109} C_VEL
LIN {X 0,Y 465.015,Z 525.096,A -85,B 0,C 180,E1 22117.497,E2 22117.497} C_VEL
LIN {X 0,Y 464.985,Z 525.123,A -85,B 0,C 180,E1 22113.844,E2 22113.844} C_VEL
LIN {X 0,Y 464.958,Z 525.093,A -85,B 0,C 180,E1 22110.215,E2 22110.215} C_VEL
LIN {X 0,Y 465,Z 525.111,A -85,B 0,C 180,E1 22106.749,E2 22106.749} C_VEL
LIN {X 0,Y 464.989,Z 525.127,A -85,B 0,C 180,E1 22103.122,E2 22103.122} C_VEL
LIN {X 0,Y 465.001,Z 525.341,A -85,B 0,C 180,E1 22102.26,E2 22102.26} C_VEL
LIN {X 0,Y 466.133,Z 528.402,A -85,B 0,C 180,E1 22102.003,E2 22102.003} C_VEL
LIN {X 0,Y 468.658,Z 530.908,A -85,B 0,C 180,E1 22101.545,E2 22101.545} C_VEL
LIN {X 0,Y 469.484,Z 531.973,A -85,B 0,C 180,E1 22101.391,E2 22101.391} C_VEL
LIN {X 0,Y 472.233,Z 535.828,A -85,B 0,C 180,E1 22100.879,E2 22100.879} C_VEL
LIN {X 0,Y 473.711,Z 537.635,A -85,B 0,C 180,E1 22100.615,E2 22100.615} C_VEL
LIN {X 0,Y 477.035,Z 541.908,A -85,B 0,C 180,E1 22100.027,E2 22100.027} C_VEL
LIN {X 0,Y 489.111,Z 558.484,A -85,B 0,C 180,E1 22097.992,E2 22097.992} C_VEL
LIN {X 0,Y 499.26,Z 573.123,A -85,B 0,C 180,E1 22096.4,E2 22096.4} C_VEL
LIN {X 0,Y 495.754,Z 713.015,A -85,B 0,C 180,E1 22093.988,E2 22093.988} C_VEL
LIN {X 0,Y 494.876,Z 720.715,A -85,B 0,C 180,E1 22093.935,E2 22093.935} C_VEL
LIN {X 0,Y 489.872,Z 741.33,A -85,B 0,C 180,E1 22094.092,E2 22094.092} C_VEL
LIN {X 0,Y 489.157,Z 747.941,A -85,B 0,C 180,E1 22094.041,E2 22094.041} C_VEL
LIN {X 0,Y 486.07,Z 864.064,A -85,B 0,C 180,E1 22092.034,E2 22092.034} C_VEL
LIN {X 0,Y 484.756,Z 886.708,A -85,B 0,C 180,E1 22091.456,E2 22091.456} C_VEL
LIN {X 0,Y 483.183,Z 907.495,A -85,B 0,C 180,E1 22090.739,E2 22090.739} C_VEL
LIN {X 0,Y 481.048,Z 929.556,A -85,B 0,C 180,E1 22089.758,E2 22089.758} C_VEL
LIN {X 0,Y 478.778,Z 950.03,A -85,B 0,C 180,E1 22088.64,E2 22088.64} C_VEL
LIN {X 0,Y 476.152,Z 970.669,A -85,B 0,C 180,E1 22087.264,E2 22087.264} C_VEL
LIN {X 0,Y 473.513,Z 990.313,A -85,B 0,C 180,E1 22085.722,E2 22085.722} C_VEL
LIN {X 0,Y 470.699,Z 1009.212,A -85,B 0,C 180,E1 22083.964,E2 22083.964} C_VEL
LIN {X 0,Y 467.954,Z 1027.614,A -85,B 0,C 180,E1 22081.978,E2 22081.978} C_VEL
LIN {X 0,Y 465.168,Z 1046.343,A -85,B 0,C 180,E1 22079.629,E2 22079.629} C_VEL
LIN {X 0,Y 462.98,Z 1061.702,A -85,B 0,C 180,E1 22077.387,E2 22077.387} C_VEL
LIN {X 0,Y 461.042,Z 1076.236,A -85,B 0,C 180,E1 22074.972,E2 22074.972} C_VEL
LIN {X 0,Y 459.461,Z 1088.865,A -85,B 0,C 180,E1 22072.52,E2 22072.52} C_VEL
LIN {X 0,Y 458.14,Z 1101.12,A -85,B 0,C 180,E1 22069.772,E2 22069.772} C_VEL
LIN {X 0,Y 457.239,Z 1110.905,A -85,B 0,C 180,E1 22067.17,E2 22067.17} C_VEL
LIN {X 0,Y 456.552,Z 1120.221,A -85,B 0,C 180,E1 22064.199,E2 22064.199} C_VEL
LIN {X 0,Y 456.202,Z 1127.059,A -85,B 0,C 180,E1 22061.505,E2 22061.505} C_VEL
LIN {X 0,Y 456.008,Z 1132.768,A -85,B 0,C 180,E1 22058.575,E2 22058.575} C_VEL
LIN {X 0,Y 455.912,Z 1136.539,A -85,B 0,C 180,E1 22055.917,E2 22055.917} C_VEL
LIN {X 0,Y 455.885,Z 1138.96,A -85,B 0,C 180,E1 22053.143,E2 22053.143} C_VEL
LIN {X 0,Y 455.887,Z 1139.886,A -85,B 0,C 180,E1 22050.629,E2 22050.629} C_VEL
LIN {X 0,Y 455.913,Z 1139.484,A -85,B 0,C 180,E1 22047.738,E2 22047.738} C_VEL
LIN {X 0,Y 455.912,Z 1137.655,A -85,B 0,C 180,E1 22045.094,E2 22045.094} C_VEL
LIN {X 0,Y 455.969,Z 1134.155,A -85,B 0,C 180,E1 22042.186,E2 22042.186} C_VEL
LIN {X 0,Y 456.086,Z 1129.663,A -85,B 0,C 180,E1 22039.644,E2 22039.644} C_VEL
LIN {X 0,Y 456.39,Z 1123.296,A -85,B 0,C 180,E1 22036.83,E2 22036.83} C_VEL
LIN {X 0,Y 456.893,Z 1115.478,A -85,B 0,C 180,E1 22034.125,E2 22034.125} C_VEL
LIN {X 0,Y 457.725,Z 1105.585,A -85,B 0,C 180,E1 22031.27,E2 22031.27} C_VEL
LIN {X 0,Y 458.813,Z 1094.761,A -85,B 0,C 180,E1 22028.658,E2 22028.658} C_VEL
LIN {X 0,Y 460.373,Z 1081.376,A -85,B 0,C 180,E1 22025.902,E2 22025.902} C_VEL
LIN {X 0,Y 462.122,Z 1068.049,A -85,B 0,C 180,E1 22023.532,E2 22023.532} C_VEL
LIN {X 0,Y 464.266,Z 1052.549,A -85,B 0,C 180,E1 22021.157,E2 22021.157} C_VEL
LIN {X 0,Y 466.716,Z 1035.803,A -85,B 0,C 180,E1 22018.916,E2 22018.916} C_VEL
LIN {X 0,Y 469.277,Z 1018.798,A -85,B 0,C 180,E1 22016.945,E2 22016.945} C_VEL
LIN {X 0,Y 472.086,Z 999.956,A -85,B 0,C 180,E1 22015.05,E2 22015.05} C_VEL
LIN {X 0,Y 474.666,Z 981.692,A -85,B 0,C 180,E1 22013.482,E2 22013.482} C_VEL
LIN {X 0,Y 477.496,Z 960.447,A -85,B 0,C 180,E1 22011.937,E2 22011.937} C_VEL
LIN {X 0,Y 479.664,Z 942.381,A -85,B 0,C 180,E1 22010.832,E2 22010.832} C_VEL
LIN {X 0,Y 481.982,Z 920.282,A -85,B 0,C 180,E1 22009.709,E2 22009.709} C_VEL
LIN {X 0,Y 483.819,Z 899.245,A -85,B 0,C 180,E1 22008.861,E2 22008.861} C_VEL
LIN {X 0,Y 485.441,Z 875.858,A -85,B 0,C 180,E1 22008.153,E2 22008.153} C_VEL
LIN {X 0,Y 486.472,Z 853.763,A -85,B 0,C 180,E1 22007.679,E2 22007.679} C_VEL
LIN {X 0,Y 491.701,Z 650.412,A -85,B 0,C 180,E1 22004.183,E2 22004.183} C_VEL
LIN {X 0,Y 493.556,Z 576.685,A -85,B 0,C 180,E1 22002.877,E2 22002.877} C_VEL
LIN {X 0,Y 480.572,Z 558.115,A -85,B 0,C 180,E1 22000.751,E2 22000.751} C_VEL
LIN {X 0,Y 472.605,Z 547.506,A -85,B 0,C 180,E1 21999.358,E2 21999.358} C_VEL
LIN {X 0,Y 468.575,Z 542.185,A -85,B 0,C 180,E1 21998.62,E2 21998.62} C_VEL
LIN {X 0,Y 465.023,Z 537.49,A -85,B 0,C 180,E1 21997.948,E2 21997.948} C_VEL
LIN {X 0,Y 462.099,Z 533.959,A -85,B 0,C 180,E1 21997.387,E2 21997.387} C_VEL
LIN {X 0,Y 461.006,Z 532.052,A -85,B 0,C 180,E1 21997.159,E2 21997.159} C_VEL
LIN {X 0,Y 458.271,Z 529.508,A -85,B 0,C 180,E1 21996.636,E2 21996.636} C_VEL
LIN {X 0,Y 457.062,Z 526.455,A -85,B 0,C 180,E1 21996.35,E2 21996.35} C_VEL
LIN {X 0,Y 457.01,Z 526.11,A -85,B 0,C 180,E1 21996.297,E2 21996.297} C_VEL
LIN {X 0,Y 457.056,Z 526.105,A -85,B 0,C 180,E1 21992.707,E2 21992.707} C_VEL
LIN {X 0,Y 457.043,Z 526.077,A -85,B 0,C 180,E1 21989.2,E2 21989.2} C_VEL
LIN {X 0,Y 457.027,Z 526.112,A -85,B 0,C 180,E1 21985.664,E2 21985.664} C_VEL
LIN {X 0,Y 457.048,Z 526.091,A -85,B 0,C 180,E1 21981.968,E2 21981.968} C_VEL
LIN {X 0,Y 457.074,Z 526.081,A -85,B 0,C 180,E1 21978.361,E2 21978.361} C_VEL
LIN {X 0,Y 457.052,Z 526.105,A -85,B 0,C 180,E1 21974.701,E2 21974.701} C_VEL
LIN {X 0,Y 457.043,Z 526.11,A -85,B 0,C 180,E1 21970.972,E2 21970.972} C_VEL
LIN {X 0,Y 457.068,Z 526.111,A -85,B 0,C 180,E1 21967.289,E2 21967.289} C_VEL
LIN {X 0,Y 457.071,Z 526.111,A -85,B 0,C 180,E1 21963.637,E2 21963.637} C_VEL
LIN {X 0,Y 457.077,Z 526.108,A -85,B 0,C 180,E1 21959.875,E2 21959.875} C_VEL
LIN {X 0,Y 457.061,Z 526.11,A -85,B 0,C 180,E1 21956.112,E2 21956.112} C_VEL
LIN {X 0,Y 457.067,Z 526.111,A -85,B 0,C 180,E1 21952.332,E2 21952.332} C_VEL
LIN {X 0,Y 457.06,Z 526.068,A -85,B 0,C 180,E1 21948.646,E2 21948.646} C_VEL
LIN {X 0,Y 457.059,Z 526.112,A -85,B 0,C 180,E1 21944.911,E2 21944.911} C_VEL
LIN {X 0,Y 457.068,Z 526.079,A -85,B 0,C 180,E1 21941.242,E2 21941.242} C_VEL
LIN {X 0,Y 457.074,Z 526.091,A -85,B 0,C 180,E1 21937.628,E2 21937.628} C_VEL
LIN {X 0,Y 457.053,Z 526.115,A -85,B 0,C 180,E1 21933.915,E2 21933.915} C_VEL
LIN {X 0,Y 457.041,Z 526.084,A -85,B 0,C 180,E1 21930.225,E2 21930.225} C_VEL
LIN {X 0,Y 457.069,Z 526.083,A -85,B 0,C 180,E1 21926.683,E2 21926.683} C_VEL
LIN {X 0,Y 457.075,Z 526.222,A -85,B 0,C 180,E1 21925.232,E2 21925.232} C_VEL
LIN {X 0,Y 458.203,Z 529.305,A -85,B 0,C 180,E1 21924.672,E2 21924.672} C_VEL
LIN {X 0,Y 459.639,Z 531.396,A -85,B 0,C 180,E1 21924.186,E2 21924.186} C_VEL
LIN {X 0,Y 461.556,Z 535.187,A -85,B 0,C 180,E1 21923.436,E2 21923.436} C_VEL
LIN {X 0,Y 463.695,Z 539.183,A -85,B 0,C 180,E1 21922.706,E2 21922.706} C_VEL
LIN {X 0,Y 469.679,Z 547.482,A -85,B 0,C 180,E1 21921.566,E2 21921.566} C_VEL
LIN {X 0,Y 479.338,Z 561.415,A -85,B 0,C 180,E1 21919.83,E2 21919.83} C_VEL
LIN {X 0,Y 490.109,Z 577.901,A -85,B 0,C 180,E1 21918.019,E2 21918.019} C_VEL
LIN {X 0,Y 493.892,Z 584.305,A -85,B 0,C 180,E1 21917.404,E2 21917.404} C_VEL
LIN {X 0,Y 488.863,Z 777.308,A -85,B 0,C 180,E1 21914.058,E2 21914.058} C_VEL
LIN {X 0,Y 485.893,Z 891.157,A -85,B 0,C 180,E1 21912.097,E2 21912.097} C_VEL
LIN {X 0,Y 484.486,Z 914.349,A -85,B 0,C 180,E1 21911.513,E2 21911.513} C_VEL
LIN {X 0,Y 482.781,Z 936.7,A -85,B 0,C 180,E1 21910.746,E2 21910.746} C_VEL
LIN {X 0,Y 480.635,Z 958.521,A -85,B 0,C 180,E1 21909.769,E2 21909.769} C_VEL
LIN {X 0,Y 478.299,Z 979.801,A -85,B 0,C 180,E1 21908.609,E2 21908.609} C_VEL
LIN {X 0,Y 475.749,Z 1000.232,A -85,B 0,C 180,E1 21907.249,E2 21907.249} C_VEL
LIN {X 0,Y 473.021,Z 1021.069,A -85,B 0,C 180,E1 21905.616,E2 21905.616} C_VEL
LIN {X 0,Y 470.415,Z 1039.573,A -85,B 0,C 180,E1 21903.913,E2 21903.913} C_VEL
LIN {X 0,Y 467.632,Z 1059.249,A -85,B 0,C 180,E1 21901.806,E2 21901.806} C_VEL
LIN {X 0,Y 465.554,Z 1073.628,A -85,B 0,C 180,E1 21900.027,E2 21900.027} C_VEL
LIN {X 0,Y 463.179,Z 1090.288,A -85,B 0,C 180,E1 21897.653,E2 21897.653} C_VEL
LIN {X 0,Y 461.23,Z 1104.732,A -85,B 0,C 180,E1 21895.281,E2 21895.281} C_VEL
LIN {X 0,Y 459.544,Z 1118.193,A -85,B 0,C 180,E1 21892.704,E2 21892.704} C_VEL
LIN {X 0,Y 458.239,Z 1130.253,A -85,B 0,C 180,E1 21890.033,E2 21890.033} C_VEL
LIN {X 0,Y 457.304,Z 1140.145,A -85,B 0,C 180,E1 21887.43,E2 21887.43} C_VEL
LIN {X 0,Y 456.62,Z 1149.321,A -85,B 0,C 180,E1 21884.571,E2 21884.571} C_VEL
LIN {X 0,Y 456.237,Z 1156.259,A -85,B 0,C 180,E1 21881.888,E2 21881.888} C_VEL
LIN {X 0,Y 456.027,Z 1162.223,A -85,B 0,C 180,E1 21878.955,E2 21878.955} C_VEL
LIN {X 0,Y 455.932,Z 1166.119,A -85,B 0,C 180,E1 21876.295,E2 21876.295} C_VEL
LIN {X 0,Y 455.888,Z 1168.849,A -85,B 0,C 180,E1 21873.395,E2 21873.395} C_VEL
LIN {X 0,Y 455.888,Z 1169.849,A -85,B 0,C 180,E1 21870.879,E2 21870.879} C_VEL
LIN {X 0,Y 455.906,Z 1169.658,A -85,B 0,C 180,E1 21868.115,E2 21868.115} C_VEL
LIN {X 0,Y 455.91,Z 1167.841,A -85,B 0,C 180,E1 21865.345,E2 21865.345} C_VEL
LIN {X 0,Y 455.943,Z 1164.68,A -85,B 0,C 180,E1 21862.566,E2 21862.566} C_VEL
LIN {X 0,Y 456.076,Z 1159.827,A -85,B 0,C 180,E1 21859.771,E2 21859.771} C_VEL
LIN {X 0,Y 456.352,Z 1153.827,A -85,B 0,C 180,E1 21857.086,E2 21857.086} C_VEL
LIN {X 0,Y 456.872,Z 1145.742,A -85,B 0,C 180,E1 21854.254,E2 21854.254} C_VEL
LIN {X 0,Y 457.678,Z 1136.175,A -85,B 0,C 180,E1 21851.463,E2 21851.463} C_VEL
LIN {X 0,Y 458.77,Z 1125.143,A -85,B 0,C 180,E1 21848.79,E2 21848.79} C_VEL
LIN {X 0,Y 460.315,Z 1111.843,A -85,B 0,C 180,E1 21846.034,E2 21846.034} C_VEL
LIN {X 0,Y 462.091,Z 1098.246,A -85,B 0,C 180,E1 21843.61,E2 21843.61} C_VEL
LIN {X 0,Y 464.234,Z 1082.766,A -85,B 0,C 180,E1 21841.233,E2 21841.233} C_VEL
LIN {X 0,Y 466.612,Z 1066.526,A -85,B 0,C 180,E1 21839.051,E2 21839.051} C_VEL
LIN {X 0,Y 469.121,Z 1048.766,A -85,B 0,C 180,E1 21837.032,E2 21837.032} C_VEL
LIN {X 0,Y 471.786,Z 1029.973,A -85,B 0,C 180,E1 21835.169,E2 21835.169} C_VEL
LIN {X 0,Y 474.396,Z 1010.626,A -85,B 0,C 180,E1 21833.533,E2 21833.533} C_VEL
LIN {X 0,Y 477.194,Z 988.919,A -85,B 0,C 180,E1 21831.974,E2 21831.974} C_VEL
LIN {X 0,Y 479.449,Z 969.602,A -85,B 0,C 180,E1 21830.81,E2 21830.81} C_VEL
LIN {X 0,Y 481.844,Z 946.168,A -85,B 0,C 180,E1 21829.652,E2 21829.652} C_VEL
LIN {X 0,Y 483.783,Z 924.424,A -85,B 0,C 180,E1 21828.805,E2 21828.805} C_VEL
LIN {X 0,Y 485.299,Z 902.139,A -85,B 0,C 180,E1 21828.157,E2 21828.157} C_VEL
LIN {X 0,Y 486.357,Z 879.205,A -85,B 0,C 180,E1 21827.676,E2 21827.676} C_VEL
LIN {X 0,Y 491.372,Z 678.592,A -85,B 0,C 180,E1 21824.24,E2 21824.24} C_VEL
LIN {X 0,Y 493.802,Z 583.805,A -85,B 0,C 180,E1 21822.575,E2 21822.575} C_VEL
LIN {X 0,Y 481.05,Z 563.83,A -85,B 0,C 180,E1 21820.467,E2 21820.467} C_VEL
LIN {X 0,Y 468.023,Z 545.009,A -85,B 0,C 180,E1 21818.126,E2 21818.126} C_VEL
LIN {X 0,Y 463.145,Z 538.434,A -85,B 0,C 180,E1 21817.191,E2 21817.191} C_VEL
LIN {X 0,Y 461.534,Z 535.167,A -85,B 0,C 180,E1 21816.566,E2 21816.566} C_VEL
LIN {X 0,Y 459.623,Z 531.352,A -85,B 0,C 180,E1 21815.815,E2 21815.815} C_VEL
LIN {X 0,Y 457.312,Z 527.292,A -85,B 0,C 180,E1 21814.947,E2 21814.947} C_VEL
LIN {X 0,Y 457.054,Z 526.083,A -85,B 0,C 180,E1 21814.741,E2 21814.741} C_VEL
LIN {X 0,Y 457.078,Z 526.103,A -85,B 0,C 180,E1 21811.081,E2 21811.081} C_VEL
LIN {X 0,Y 457.05,Z 526.101,A -85,B 0,C 180,E1 21807.489,E2 21807.489} C_VEL
LIN {X 0,Y 457.043,Z 526.071,A -85,B 0,C 180,E1 21803.736,E2 21803.736} C_VEL
LIN {X 0,Y 457.07,Z 526.107,A -85,B 0,C 180,E1 21800.086,E2 21800.086} C_VEL
LIN {X 0,Y 457.067,Z 526.077,A -85,B 0,C 180,E1 21796.391,E2 21796.391} C_VEL
LIN {X 0,Y 457.064,Z 526.096,A -85,B 0,C 180,E1 21792.764,E2 21792.764} C_VEL
LIN {X 0,Y 457.059,Z 526.095,A -85,B 0,C 180,E1 21789.062,E2 21789.062} C_VEL
LIN {X 0,Y 457.069,Z 526.101,A -85,B 0,C 180,E1 21785.397,E2 21785.397} C_VEL
LIN {X 0,Y 457.059,Z 526.106,A -85,B 0,C 180,E1 21781.629,E2 21781.629} C_VEL
LIN {X 0,Y 457.069,Z 526.104,A -85,B 0,C 180,E1 21777.994,E2 21777.994} C_VEL
LIN {X 0,Y 457.071,Z 526.102,A -85,B 0,C 180,E1 21774.224,E2 21774.224} C_VEL
LIN {X 0,Y 457.063,Z 526.079,A -85,B 0,C 180,E1 21770.557,E2 21770.557} C_VEL
LIN {X 0,Y 457.046,Z 526.111,A -85,B 0,C 180,E1 21766.849,E2 21766.849} C_VEL
LIN {X 0,Y 457.051,Z 526.072,A -85,B 0,C 180,E1 21763.216,E2 21763.216} C_VEL
LIN {X 0,Y 457.078,Z 526.112,A -85,B 0,C 180,E1 21759.512,E2 21759.512} C_VEL
LIN {X 0,Y 457.05,Z 526.071,A -85,B 0,C 180,E1 21755.852,E2 21755.852} C_VEL
LIN {X 0,Y 457.027,Z 526.109,A -85,B 0,C 180,E1 21752.225,E2 21752.225} C_VEL
LIN {X 0,Y 457.041,Z 526.105,A -85,B 0,C 180,E1 21748.562,E2 21748.562} C_VEL
LIN {X 0,Y 457.063,Z 526.078,A -85,B 0,C 180,E1 21745.03,E2 21745.03} C_VEL
LIN {X 0,Y 457.041,Z 526.266,A -85,B 0,C 180,E1 21743.559,E2 21743.559} C_VEL
LIN {X 0,Y 458.202,Z 529.384,A -85,B 0,C 180,E1 21743.28,E2 21743.28} C_VEL
LIN {X 0,Y 460.932,Z 532.009,A -85,B 0,C 180,E1 21742.756,E2 21742.756} C_VEL
LIN {X 0,Y 464.113,Z 536.655,A -85,B 0,C 180,E1 21742.121,E2 21742.121} C_VEL
LIN {X 0,Y 466.055,Z 538.732,A -85,B 0,C 180,E1 21741.761,E2 21741.761} C_VEL
LIN {X 0,Y 471.001,Z 545.463,A -85,B 0,C 180,E1 21740.836,E2 21740.836} C_VEL
LIN {X 0,Y 475.367,Z 551.151,A -85,B 0,C 180,E1 21740.055,E2 21740.055} C_VEL
LIN {X 0,Y 485.156,Z 564.589,A -85,B 0,C 180,E1 21738.385,E2 21738.385} C_VEL
LIN {X 0,Y 493.679,Z 577.009,A -85,B 0,C 180,E1 21737.01,E2 21737.01} C_VEL
LIN {X 0,Y 489.157,Z 747.941,A -85,B 0,C 180,E1 21734.041,E2 21734.041} C_VEL
LIN {X 0,Y 488.241,Z 755.641,A -85,B 0,C 180,E1 21733.991,E2 21733.991} C_VEL
LIN {X 0,Y 483.217,Z 776.243,A -85,B 0,C 180,E1 21734.153,E2 21734.153} C_VEL
LIN {X 0,Y 482.498,Z 782.85,A -85,B 0,C 180,E1 21734.102,E2 21734.102} C_VEL
LIN {X 0,Y 480.131,Z 865.195,A -85,B 0,C 180,E1 21732.657,E2 21732.657} C_VEL
LIN {X 0,Y 478.74,Z 887.553,A -85,B 0,C 180,E1 21732.075,E2 21732.075} C_VEL
LIN {X 0,Y 477.031,Z 908.984,A -85,B 0,C 180,E1 21731.325,E2 21731.325} C_VEL
LIN {X 0,Y 474.807,Z 930.493,A -85,B 0,C 180,E1 21730.349,E2 21730.349} C_VEL
LIN {X 0,Y 472.352,Z 951.458,A -85,B 0,C 180,E1 21729.188,E2 21729.188} C_VEL
LIN {X 0,Y 469.615,Z 971.596,A -85,B 0,C 180,E1 21727.821,E2 21727.821} C_VEL
LIN {X 0,Y 466.781,Z 991.357,A -85,B 0,C 180,E1 21726.243,E2 21726.243} C_VEL
LIN {X 0,Y 463.918,Z 1009.528,A -85,B 0,C 180,E1 21724.53,E2 21724.53} C_VEL
LIN {X 0,Y 461.005,Z 1027.77,A -85,B 0,C 180,E1 21722.54,E2 21722.54} C_VEL
LIN {X 0,Y 458.415,Z 1043.764,A -85,B 0,C 180,E1 21720.51,E2 21720.51} C_VEL
LIN {X 0,Y 455.592,Z 1061.705,A -85,B 0,C 180,E1 21717.87,E2 21717.87} C_VEL
LIN {X 0,Y 453.536,Z 1076.004,A -85,B 0,C 180,E1 21715.461,E2 21715.461} C_VEL
LIN {X 0,Y 451.799,Z 1088.868,A -85,B 0,C 180,E1 21712.924,E2 21712.924} C_VEL
LIN {X 0,Y 450.363,Z 1101.122,A -85,B 0,C 180,E1 21710.128,E2 21710.128} C_VEL
LIN {X 0,Y 449.375,Z 1110.907,A -85,B 0,C 180,E1 21707.481,E2 21707.481} C_VEL
LIN {X 0,Y 448.625,Z 1120.223,A -85,B 0,C 180,E1 21704.455,E2 21704.455} C_VEL
LIN {X 0,Y 448.25,Z 1126.758,A -85,B 0,C 180,E1 21701.842,E2 21701.842} C_VEL
LIN {X 0,Y 448.029,Z 1132.563,A -85,B 0,C 180,E1 21698.858,E2 21698.858} C_VEL
LIN {X 0,Y 447.931,Z 1136.221,A -85,B 0,C 180,E1 21696.28,E2 21696.28} C_VEL
LIN {X 0,Y 447.888,Z 1138.892,A -85,B 0,C 180,E1 21693.328,E2 21693.328} C_VEL
LIN {X 0,Y 447.888,Z 1139.863,A -85,B 0,C 180,E1 21690.768,E2 21690.768} C_VEL
LIN {X 0,Y 447.909,Z 1139.619,A -85,B 0,C 180,E1 21687.953,E2 21687.953} C_VEL
LIN {X 0,Y 447.909,Z 1137.882,A -85,B 0,C 180,E1 21685.263,E2 21685.263} C_VEL
LIN {X 0,Y 447.94,Z 1134.897,A -85,B 0,C 180,E1 21682.562,E2 21682.562} C_VEL
LIN {X 0,Y 448.083,Z 1130.17,A -85,B 0,C 180,E1 21679.717,E2 21679.717} C_VEL
LIN {X 0,Y 448.357,Z 1124.544,A -85,B 0,C 180,E1 21677.115,E2 21677.115} C_VEL
LIN {X 0,Y 448.908,Z 1116.58,A -85,B 0,C 180,E1 21674.197,E2 21674.197} C_VEL
LIN {X 0,Y 449.71,Z 1107.542,A -85,B 0,C 180,E1 21671.462,E2 21671.462} C_VEL
LIN {X 0,Y 450.893,Z 1096.362,A -85,B 0,C 180,E1 21668.647,E2 21668.647} C_VEL
LIN {X 0,Y 452.427,Z 1084.172,A -85,B 0,C 180,E1 21666.006,E2 21666.006} C_VEL
LIN {X 0,Y 454.317,Z 1070.354,A -85,B 0,C 180,E1 21663.464,E2 21663.464} C_VEL
LIN {X 0,Y 456.85,Z 1053.521,A -85,B 0,C 180,E1 21660.787,E2 21660.787} C_VEL
LIN {X 0,Y 459.322,Z 1038.155,A -85,B 0,C 180,E1 21658.65,E2 21658.65} C_VEL
LIN {X 0,Y 462.098,Z 1020.961,A -85,B 0,C 180,E1 21656.594,E2 21656.594} C_VEL
LIN {X 0,Y 464.977,Z 1003.076,A -85,B 0,C 180,E1 21654.735,E2 21654.735} C_VEL
LIN {X 0,Y 467.889,Z 983.596,A -85,B 0,C 180,E1 21653.019,E2 21653.019} C_VEL
LIN {X 0,Y 470.766,Z 963.592,A -85,B 0,C 180,E1 21651.516,E2 21651.516} C_VEL
LIN {X 0,Y 473.23,Z 944.185,A -85,B 0,C 180,E1 21650.3,E2 21650.3} C_VEL
LIN {X 0,Y 475.609,Z 923.434,A -85,B 0,C 180,E1 21649.211,E2 21649.211} C_VEL
LIN {X 0,Y 477.62,Z 901.542,A -85,B 0,C 180,E1 21648.302,E2 21648.302} C_VEL
LIN {X 0,Y 479.405,Z 877.744,A -85,B 0,C 180,E1 21647.554,E2 21647.554} C_VEL
LIN {X 0,Y 480.498,Z 856.083,A -85,B 0,C 180,E1 21647.076,E2 21647.076} C_VEL
LIN {X 0,Y 486.05,Z 654.175,A -85,B 0,C 180,E1 21643.567,E2 21643.567} C_VEL
LIN {X 0,Y 488.01,Z 580.545,A -85,B 0,C 180,E1 21642.248,E2 21642.248} C_VEL
LIN {X 0,Y 476.469,Z 563.981,A -85,B 0,C 180,E1 21640.305,E2 21640.305} C_VEL
LIN {X 0,Y 468.73,Z 553.577,A -85,B 0,C 180,E1 21638.918,E2 21638.918} C_VEL
LIN {X 0,Y 464.47,Z 547.955,A -85,B 0,C 180,E1 21638.118,E2 21638.118} C_VEL
LIN {X 0,Y 461.498,Z 544.011,A -85,B 0,C 180,E1 21637.542,E2 21637.542} C_VEL
LIN {X 0,Y 458.232,Z 539.729,A -85,B 0,C 180,E1 21636.893,E2 21636.893} C_VEL
LIN {X 0,Y 456.686,Z 538.067,A -85,B 0,C 180,E1 21636.588,E2 21636.588} C_VEL
LIN {X 0,Y 453.958,Z 534.401,A -85,B 0,C 180,E1 21636.021,E2 21636.021} C_VEL
LIN {X 0,Y 453.209,Z 533.136,A -85,B 0,C 180,E1 21635.855,E2 21635.855} C_VEL
LIN {X 0,Y 450.554,Z 530.757,A -85,B 0,C 180,E1 21635.317,E2 21635.317} C_VEL
LIN {X 0,Y 449.219,Z 527.665,A -85,B 0,C 180,E1 21634.989,E2 21634.989} C_VEL
LIN {X 0,Y 449.12,Z 527.065,A -85,B 0,C 180,E1 21634.939,E2 21634.939} C_VEL
LIN {X 0,Y 449.11,Z 527.095,A -85,B 0,C 180,E1 21631.247,E2 21631.247} C_VEL
LIN {X 0,Y 449.084,Z 527.092,A -85,B 0,C 180,E1 21627.588,E2 21627.588} C_VEL
LIN {X 0,Y 449.094,Z 527.062,A -85,B 0,C 180,E1 21623.904,E2 21623.904} C_VEL
LIN {X 0,Y 449.14,Z 527.102,A -85,B 0,C 180,E1 21620.321,E2 21620.321} C_VEL
LIN {X 0,Y 449.121,Z 527.056,A -85,B 0,C 180,E1 21616.557,E2 21616.557} C_VEL
LIN {X 0,Y 449.103,Z 527.105,A -85,B 0,C 180,E1 21612.995,E2 21612.995} C_VEL
LIN {X 0,Y 449.116,Z 527.099,A -85,B 0,C 180,E1 21609.224,E2 21609.224} C_VEL
LIN {X 0,Y 449.134,Z 527.094,A -85,B 0,C 180,E1 21605.622,E2 21605.622} C_VEL
LIN {X 0,Y 449.132,Z 527.094,A -85,B 0,C 180,E1 21601.914,E2 21601.914} C_VEL
LIN {X 0,Y 449.119,Z 527.098,A -85,B 0,C 180,E1 21598.214,E2 21598.214} C_VEL
LIN {X 0,Y 449.129,Z 527.095,A -85,B 0,C 180,E1 21594.507,E2 21594.507} C_VEL
LIN {X 0,Y 449.125,Z 527.089,A -85,B 0,C 180,E1 21590.777,E2 21590.777} C_VEL
LIN {X 0,Y 449.119,Z 527.079,A -85,B 0,C 180,E1 21587.006,E2 21587.006} C_VEL
LIN {X 0,Y 449.128,Z 527.066,A -85,B 0,C 180,E1 21583.311,E2 21583.311} C_VEL
LIN {X 0,Y 449.136,Z 527.101,A -85,B 0,C 180,E1 21579.543,E2 21579.543} C_VEL
LIN {X 0,Y 449.121,Z 527.064,A -85,B 0,C 180,E1 21575.819,E2 21575.819} C_VEL
LIN {X 0,Y 449.102,Z 527.082,A -85,B 0,C 180,E1 21572.112,E2 21572.112} C_VEL
LIN {X 0,Y 449.119,Z 527.106,A -85,B 0,C 180,E1 21568.455,E2 21568.455} C_VEL
LIN {X 0,Y 449.143,Z 527.209,A -85,B 0,C 180,E1 21566.529,E2 21566.529} C_VEL
LIN {X 0,Y 450.306,Z 530.414,A -85,B 0,C 180,E1 21565.915,E2 21565.915} C_VEL
LIN {X 0,Y 451.896,Z 532.744,A -85,B 0,C 180,E1 21565.345,E2 21565.345} C_VEL
LIN {X 0,Y 454.728,Z 538.254,A -85,B 0,C 180,E1 21564.226,E2 21564.226} C_VEL
LIN {X 0,Y 465.434,Z 552.832,A -85,B 0,C 180,E1 21562.093,E2 21562.093} C_VEL
LIN {X 0,Y 477.726,Z 570.816,A -85,B 0,C 180,E1 21559.843,E2 21559.843} C_VEL
LIN {X 0,Y 488.362,Z 587.776,A -85,B 0,C 180,E1 21558.033,E2 21558.033} C_VEL
LIN {X 0,Y 482.963,Z 782.5,A -85,B 0,C 180,E1 21554.628,E2 21554.628} C_VEL
LIN {X 0,Y 479.948,Z 890.963,A -85,B 0,C 180,E1 21552.739,E2 21552.739} C_VEL
LIN {X 0,Y 478.438,Z 914.307,A -85,B 0,C 180,E1 21552.147,E2 21552.147} C_VEL
LIN {X 0,Y 476.611,Z 936.921,A -85,B 0,C 180,E1 21551.363,E2 21551.363} C_VEL
LIN {X 0,Y 474.391,Z 958.214,A -85,B 0,C 180,E1 21550.399,E2 21550.399} C_VEL
LIN {X 0,Y 471.914,Z 979.492,A -85,B 0,C 180,E1 21549.23,E2 21549.23} C_VEL
LIN {X 0,Y 469.193,Z 999.922,A -85,B 0,C 180,E1 21547.86,E2 21547.86} C_VEL
LIN {X 0,Y 466.292,Z 1020.758,A -85,B 0,C 180,E1 21546.21,E2 21546.21} C_VEL
LIN {X 0,Y 463.571,Z 1038.922,A -85,B 0,C 180,E1 21544.521,E2 21544.521} C_VEL
LIN {X 0,Y 460.57,Z 1058.695,A -85,B 0,C 180,E1 21542.384,E2 21542.384} C_VEL
LIN {X 0,Y 458.033,Z 1075.5,A -85,B 0,C 180,E1 21540.282,E2 21540.282} C_VEL
LIN {X 0,Y 455.796,Z 1090.319,A -85,B 0,C 180,E1 21538.135,E2 21538.135} C_VEL
LIN {X 0,Y 453.704,Z 1104.73,A -85,B 0,C 180,E1 21535.731,E2 21535.731} C_VEL
LIN {X 0,Y 451.937,Z 1117.806,A -85,B 0,C 180,E1 21533.191,E2 21533.191} C_VEL
LIN {X 0,Y 450.526,Z 1129.747,A -85,B 0,C 180,E1 21530.521,E2 21530.521} C_VEL
LIN {X 0,Y 449.445,Z 1140.143,A -85,B 0,C 180,E1 21527.745,E2 21527.745} C_VEL
LIN {X 0,Y 448.703,Z 1149.285,A -85,B 0,C 180,E1 21524.848,E2 21524.848} C_VEL
LIN {X 0,Y 448.285,Z 1155.955,A -85,B 0,C 180,E1 21522.233,E2 21522.233} C_VEL
LIN {X 0,Y 448.044,Z 1161.809,A -85,B 0,C 180,E1 21519.375,E2 21519.375} C_VEL
LIN {X 0,Y 447.94,Z 1165.828,A -85,B 0,C 180,E1 21516.643,E2 21516.643} C_VEL
LIN {X 0,Y 447.906,Z 1168.676,A -85,B 0,C 180,E1 21513.778,E2 21513.778} C_VEL
LIN {X 0,Y 447.893,Z 1169.826,A -85,B 0,C 180,E1 21511.023,E2 21511.023} C_VEL
LIN {X 0,Y 447.906,Z 1169.735,A -85,B 0,C 180,E1 21508.465,E2 21508.465} C_VEL
LIN {X 0,Y 447.911,Z 1168.068,A -85,B 0,C 180,E1 21505.519,E2 21505.519} C_VEL
LIN {X 0,Y 447.931,Z 1165.319,A -85,B 0,C 180,E1 21502.948,E2 21502.948} C_VEL
LIN {X 0,Y 448.063,Z 1160.589,A -85,B 0,C 180,E1 21499.976,E2 21499.976} C_VEL
LIN {X 0,Y 448.324,Z 1155.044,A -85,B 0,C 180,E1 21497.375,E2 21497.375} C_VEL
LIN {X 0,Y 448.875,Z 1146.955,A -85,B 0,C 180,E1 21494.364,E2 21494.364} C_VEL
LIN {X 0,Y 449.629,Z 1138.284,A -85,B 0,C 180,E1 21491.719,E2 21491.719} C_VEL
LIN {X 0,Y 450.834,Z 1126.862,A -85,B 0,C 180,E1 21488.807,E2 21488.807} C_VEL
LIN {X 0,Y 452.366,Z 1114.622,A -85,B 0,C 180,E1 21486.141,E2 21486.141} C_VEL
LIN {X 0,Y 454.239,Z 1100.874,A -85,B 0,C 180,E1 21483.599,E2 21483.599} C_VEL
LIN {X 0,Y 456.473,Z 1085.891,A -85,B 0,C 180,E1 21481.181,E2 21481.181} C_VEL
LIN {X 0,Y 458.87,Z 1069.836,A -85,B 0,C 180,E1 21478.98,E2 21478.98} C_VEL
LIN {X 0,Y 461.696,Z 1051.304,A -85,B 0,C 180,E1 21476.776,E2 21476.776} C_VEL
LIN {X 0,Y 464.348,Z 1033.84,A -85,B 0,C 180,E1 21474.981,E2 21474.981} C_VEL
LIN {X 0,Y 467.286,Z 1013.594,A -85,B 0,C 180,E1 21473.193,E2 21473.193} C_VEL
LIN {X 0,Y 470.103,Z 993.557,A -85,B 0,C 180,E1 21471.684,E2 21471.684} C_VEL
LIN {X 0,Y 472.719,Z 972.712,A -85,B 0,C 180,E1 21470.378,E2 21470.378} C_VEL
LIN {X 0,Y 475.119,Z 951.738,A -85,B 0,C 180,E1 21469.278,E2 21469.278} C_VEL
LIN {X 0,Y 477.235,Z 929.188,A -85,B 0,C 180,E1 21468.347,E2 21468.347} C_VEL
LIN {X 0,Y 479.068,Z 906.072,A -85,B 0,C 180,E1 21467.618,E2 21467.618} C_VEL
LIN {X 0,Y 480.232,Z 883.973,A -85,B 0,C 180,E1 21467.127,E2 21467.127} C_VEL
LIN {X 0,Y 485.565,Z 685.936,A -85,B 0,C 180,E1 21463.692,E2 21463.692} C_VEL
LIN {X 0,Y 488.232,Z 587.358,A -85,B 0,C 180,E1 21461.942,E2 21461.942} C_VEL
LIN {X 0,Y 476.5,Z 569.068,A -85,B 0,C 180,E1 21459.947,E2 21459.947} C_VEL
LIN {X 0,Y 466.081,Z 553.861,A -85,B 0,C 180,E1 21458.04,E2 21458.04} C_VEL
LIN {X 0,Y 456.979,Z 541.303,A -85,B 0,C 180,E1 21456.249,E2 21456.249} C_VEL
LIN {X 0,Y 454.386,Z 537.543,A -85,B 0,C 180,E1 21455.67,E2 21455.67} C_VEL
LIN {X 0,Y 451.715,Z 532.127,A -85,B 0,C 180,E1 21454.559,E2 21454.559} C_VEL
LIN {X 0,Y 449.569,Z 528.939,A -85,B 0,C 180,E1 21453.78,E2 21453.78} C_VEL
LIN {X 0,Y 449.125,Z 527.07,A -85,B 0,C 180,E1 21453.435,E2 21453.435} C_VEL
LIN {X 0,Y 449.099,Z 527.066,A -85,B 0,C 180,E1 21449.767,E2 21449.767} C_VEL
LIN {X 0,Y 449.11,Z 527.099,A -85,B 0,C 180,E1 21446.013,E2 21446.013} C_VEL
LIN {X 0,Y 449.137,Z 527.071,A -85,B 0,C 180,E1 21442.237,E2 21442.237} C_VEL
LIN {X 0,Y 449.13,Z 527.06,A -85,B 0,C 180,E1 21438.49,E2 21438.49} C_VEL
LIN {X 0,Y 449.134,Z 527.099,A -85,B 0,C 180,E1 21434.701,E2 21434.701} C_VEL
LIN {X 0,Y 449.116,Z 527.055,A -85,B 0,C 180,E1 21430.908,E2 21430.908} C_VEL
LIN {X 0,Y 449.129,Z 527.102,A -85,B 0,C 180,E1 21427.161,E2 21427.161} C_VEL
LIN {X 0,Y 449.127,Z 527.101,A -85,B 0,C 180,E1 21423.446,E2 21423.446} C_VEL
LIN {X 0,Y 449.121,Z 527.101,A -85,B 0,C 180,E1 21419.745,E2 21419.745} C_VEL
LIN {X 0,Y 449.131,Z 527.101,A -85,B 0,C 180,E1 21416.042,E2 21416.042} C_VEL
LIN {X 0,Y 449.135,Z 527.102,A -85,B 0,C 180,E1 21412.324,E2 21412.324} C_VEL
LIN {X 0,Y 449.116,Z 527.059,A -85,B 0,C 180,E1 21408.572,E2 21408.572} C_VEL
LIN {X 0,Y 449.105,Z 527.097,A -85,B 0,C 180,E1 21404.901,E2 21404.901} C_VEL
LIN {X 0,Y 449.114,Z 527.069,A -85,B 0,C 180,E1 21401.167,E2 21401.167} C_VEL
LIN {X 0,Y 449.138,Z 527.069,A -85,B 0,C 180,E1 21397.486,E2 21397.486} C_VEL
LIN {X 0,Y 449.117,Z 527.101,A -85,B 0,C 180,E1 21393.702,E2 21393.702} C_VEL
LIN {X 0,Y 449.082,Z 527.067,A -85,B 0,C 180,E1 21390.084,E2 21390.084} C_VEL
LIN {X 0,Y 449.092,Z 527.08,A -85,B 0,C 180,E1 21386.376,E2 21386.376} C_VEL
LIN {X 0,Y 449.159,Z 527.308,A -85,B 0,C 180,E1 21384.93,E2 21384.93} C_VEL
LIN {X 0,Y 450.353,Z 530.456,A -85,B 0,C 180,E1 21384.626,E2 21384.626} C_VEL
LIN {X 0,Y 452.854,Z 532.926,A -85,B 0,C 180,E1 21384.112,E2 21384.112} C_VEL
LIN {X 0,Y 453.709,Z 533.861,A -85,B 0,C 180,E1 21383.937,E2 21383.937} C_VEL
LIN {X 0,Y 456.208,Z 537.589,A -85,B 0,C 180,E1 21383.406,E2 21383.406} C_VEL
LIN {X 0,Y 458.165,Z 539.611,A -85,B 0,C 180,E1 21383.022,E2 21383.022} C_VEL
LIN {X 0,Y 461.428,Z 543.945,A -85,B 0,C 180,E1 21382.373,E2 21382.373} C_VEL
LIN {X 0,Y 467.423,Z 551.861,A -85,B 0,C 180,E1 21381.228,E2 21381.228} C_VEL
LIN {X 0,Y 474.212,Z 560.88,A -85,B 0,C 180,E1 21379.998,E2 21379.998} C_VEL
LIN {X 0,Y 486.622,Z 578.383,A -85,B 0,C 180,E1 21377.889,E2 21377.889} C_VEL
LIN {X 0,Y 488.151,Z 581.07,A -85,B 0,C 180,E1 21377.631,E2 21377.631} C_VEL
LIN {X 0,Y 482.498,Z 782.85,A -85,B 0,C 180,E1 21374.102,E2 21374.102} C_VEL
LIN {X 0,Y 481.574,Z 790.55,A -85,B 0,C 180,E1 21374.052,E2 21374.052} C_VEL
LIN {X 0,Y 476.534,Z 811.143,A -85,B 0,C 180,E1 21374.22,E2 21374.22} C_VEL
LIN {X 0,Y 475.807,Z 817.75,A -85,B 0,C 180,E1 21374.169,E2 21374.169} C_VEL
LIN {X 0,Y 474.205,Z 867.379,A -85,B 0,C 180,E1 21373.273,E2 21373.273} C_VEL
LIN {X 0,Y 472.733,Z 889.046,A -85,B 0,C 180,E1 21372.689,E2 21372.689} C_VEL
LIN {X 0,Y 470.862,Z 911.051,A -85,B 0,C 180,E1 21371.9,E2 21371.9} C_VEL
LIN {X 0,Y 468.554,Z 931.96,A -85,B 0,C 180,E1 21370.929,E2 21370.929} C_VEL
LIN {X 0,Y 465.956,Z 952.793,A -85,B 0,C 180,E1 21369.752,E2 21369.752} C_VEL
LIN {X 0,Y 463.048,Z 973.044,A -85,B 0,C 180,E1 21368.354,E2 21368.354} C_VEL
LIN {X 0,Y 459.841,Z 993.853,A -85,B 0,C 180,E1 21366.646,E2 21366.646} C_VEL
LIN {X 0,Y 456.967,Z 1011.162,A -85,B 0,C 180,E1 21364.979,E2 21364.979} C_VEL
LIN {X 0,Y 453.693,Z 1030.274,A -85,B 0,C 180,E1 21362.83,E2 21362.83} C_VEL
LIN {X 0,Y 450.811,Z 1047.176,A -85,B 0,C 180,E1 21360.621,E2 21360.621} C_VEL
LIN {X 0,Y 448.101,Z 1063.002,A -85,B 0,C 180,E1 21358.191,E2 21358.191} C_VEL
LIN {X 0,Y 445.69,Z 1078.115,A -85,B 0,C 180,E1 21355.515,E2 21355.515} C_VEL
LIN {X 0,Y 443.981,Z 1090.14,A -85,B 0,C 180,E1 21353.07,E2 21353.07} C_VEL
LIN {X 0,Y 442.465,Z 1102.153,A -85,B 0,C 180,E1 21350.227,E2 21350.227} C_VEL
LIN {X 0,Y 441.431,Z 1111.852,A -85,B 0,C 180,E1 21347.525,E2 21347.525} C_VEL
LIN {X 0,Y 440.673,Z 1120.577,A -85,B 0,C 180,E1 21344.588,E2 21344.588} C_VEL
LIN {X 0,Y 440.256,Z 1127.365,A -85,B 0,C 180,E1 21341.795,E2 21341.795} C_VEL
LIN {X 0,Y 440.034,Z 1132.771,A -85,B 0,C 180,E1 21338.889,E2 21338.889} C_VEL
LIN {X 0,Y 439.931,Z 1136.382,A -85,B 0,C 180,E1 21336.263,E2 21336.263} C_VEL
LIN {X 0,Y 439.887,Z 1138.96,A -85,B 0,C 180,E1 21333.258,E2 21333.258} C_VEL
LIN {X 0,Y 439.889,Z 1139.863,A -85,B 0,C 180,E1 21330.782,E2 21330.782} C_VEL
LIN {X 0,Y 439.91,Z 1139.618,A -85,B 0,C 180,E1 21327.916,E2 21327.916} C_VEL
LIN {X 0,Y 439.91,Z 1137.881,A -85,B 0,C 180,E1 21325.176,E2 21325.176} C_VEL
LIN {X 0,Y 439.951,Z 1134.896,A -85,B 0,C 180,E1 21322.426,E2 21322.426} C_VEL
LIN {X 0,Y 440.112,Z 1130.168,A -85,B 0,C 180,E1 21319.529,E2 21319.529} C_VEL
LIN {X 0,Y 440.407,Z 1124.542,A -85,B 0,C 180,E1 21316.878,E2 21316.878} C_VEL
LIN {X 0,Y 440.996,Z 1116.687,A -85,B 0,C 180,E1 21313.942,E2 21313.942} C_VEL
LIN {X 0,Y 441.883,Z 1107.54,A -85,B 0,C 180,E1 21311.121,E2 21311.121} C_VEL
LIN {X 0,Y 443.156,Z 1096.47,A -85,B 0,C 180,E1 21308.283,E2 21308.283} C_VEL
LIN {X 0,Y 444.846,Z 1084.046,A -85,B 0,C 180,E1 21305.547,E2 21305.547} C_VEL
LIN {X 0,Y 447.289,Z 1068.011,A -85,B 0,C 180,E1 21302.554,E2 21302.554} C_VEL
LIN {X 0,Y 449.842,Z 1052.634,A -85,B 0,C 180,E1 21300.095,E2 21300.095} C_VEL
LIN {X 0,Y 452.665,Z 1036.408,A -85,B 0,C 180,E1 21297.837,E2 21297.837} C_VEL
LIN {X 0,Y 455.569,Z 1019.4,A -85,B 0,C 180,E1 21295.816,E2 21295.816} C_VEL
LIN {X 0,Y 458.738,Z 1000.521,A -85,B 0,C 180,E1 21293.873,E2 21293.873} C_VEL
LIN {X 0,Y 461.66,Z 982.283,A -85,B 0,C 180,E1 21292.278,E2 21292.278} C_VEL
LIN {X 0,Y 464.828,Z 960.895,A -85,B 0,C 180,E1 21290.693,E2 21290.693} C_VEL
LIN {X 0,Y 467.361,Z 941.839,A -85,B 0,C 180,E1 21289.511,E2 21289.511} C_VEL
LIN {X 0,Y 469.948,Z 919.305,A -85,B 0,C 180,E1 21288.368,E2 21288.368} C_VEL
LIN {X 0,Y 472.139,Z 896.926,A -85,B 0,C 180,E1 21287.474,E2 21287.474} C_VEL
LIN {X 0,Y 473.711,Z 875.101,A -85,B 0,C 180,E1 21286.828,E2 21286.828} C_VEL
LIN {X 0,Y 474.85,Z 851.932,A -85,B 0,C 180,E1 21286.334,E2 21286.334} C_VEL
LIN {X 0,Y 480.785,Z 647.516,A -85,B 0,C 180,E1 21282.754,E2 21282.754} C_VEL
LIN {X 0,Y 482.569,Z 584.366,A -85,B 0,C 180,E1 21281.61,E2 21281.61} C_VEL
LIN {X 0,Y 469.465,Z 565.629,A -85,B 0,C 180,E1 21279.317,E2 21279.317} C_VEL
LIN {X 0,Y 458.274,Z 550.758,A -85,B 0,C 180,E1 21277.183,E2 21277.183} C_VEL
LIN {X 0,Y 454.651,Z 545.954,A -85,B 0,C 180,E1 21276.445,E2 21276.445} C_VEL
LIN {X 0,Y 450.922,Z 541.508,A -85,B 0,C 180,E1 21275.674,E2 21275.674} C_VEL
LIN {X 0,Y 449.651,Z 539.777,A -85,B 0,C 180,E1 21275.398,E2 21275.398} C_VEL
LIN {X 0,Y 446.72,Z 536.402,A -85,B 0,C 180,E1 21274.767,E2 21274.767} C_VEL
LIN {X 0,Y 445.648,Z 534.292,A -85,B 0,C 180,E1 21274.508,E2 21274.508} C_VEL
LIN {X 0,Y 442.804,Z 532.044,A -85,B 0,C 180,E1 21273.899,E2 21273.899} C_VEL
LIN {X 0,Y 441.332,Z 529.037,A -85,B 0,C 180,E1 21273.524,E2 21273.524} C_VEL
LIN {X 0,Y 441.157,Z 528.064,A -85,B 0,C 180,E1 21273.418,E2 21273.418} C_VEL
LIN {X 0,Y 441.138,Z 528.056,A -85,B 0,C 180,E1 21269.761,E2 21269.761} C_VEL
LIN {X 0,Y 441.162,Z 528.094,A -85,B 0,C 180,E1 21266.084,E2 21266.084} C_VEL
LIN {X 0,Y 441.199,Z 528.052,A -85,B 0,C 180,E1 21262.379,E2 21262.379} C_VEL
LIN {X 0,Y 441.183,Z 528.062,A -85,B 0,C 180,E1 21258.636,E2 21258.636} C_VEL
LIN {X 0,Y 441.161,Z 528.079,A -85,B 0,C 180,E1 21254.974,E2 21254.974} C_VEL
LIN {X 0,Y 441.171,Z 528.086,A -85,B 0,C 180,E1 21251.24,E2 21251.24} C_VEL
LIN {X 0,Y 441.202,Z 528.084,A -85,B 0,C 180,E1 21247.553,E2 21247.553} C_VEL
LIN {X 0,Y 441.193,Z 528.085,A -85,B 0,C 180,E1 21243.769,E2 21243.769} C_VEL
LIN {X 0,Y 441.192,Z 528.084,A -85,B 0,C 180,E1 21240,E2 21240} C_VEL
LIN {X 0,Y 441.183,Z 528.087,A -85,B 0,C 180,E1 21236.232,E2 21236.232} C_VEL
LIN {X 0,Y 441.195,Z 528.088,A -85,B 0,C 180,E1 21232.447,E2 21232.447} C_VEL
LIN {X 0,Y 441.182,Z 528.041,A -85,B 0,C 180,E1 21228.629,E2 21228.629} C_VEL
LIN {X 0,Y 441.181,Z 528.089,A -85,B 0,C 180,E1 21224.893,E2 21224.893} C_VEL
LIN {X 0,Y 441.188,Z 528.055,A -85,B 0,C 180,E1 21221.091,E2 21221.091} C_VEL
LIN {X 0,Y 441.193,Z 528.059,A -85,B 0,C 180,E1 21217.34,E2 21217.34} C_VEL
LIN {X 0,Y 441.194,Z 528.093,A -85,B 0,C 180,E1 21213.531,E2 21213.531} C_VEL
LIN {X 0,Y 441.158,Z 528.062,A -85,B 0,C 180,E1 21209.942,E2 21209.942} C_VEL
LIN {X 0,Y 441.192,Z 528.314,A -85,B 0,C 180,E1 21207.905,E2 21207.905} C_VEL
LIN {X 0,Y 442.632,Z 531.748,A -85,B 0,C 180,E1 21207.171,E2 21207.171} C_VEL
LIN {X 0,Y 443.972,Z 533.673,A -85,B 0,C 180,E1 21206.667,E2 21206.667} C_VEL
LIN {X 0,Y 445.974,Z 537.456,A -85,B 0,C 180,E1 21205.825,E2 21205.825} C_VEL
LIN {X 0,Y 452.007,Z 545.735,A -85,B 0,C 180,E1 21204.503,E2 21204.503} C_VEL
LIN {X 0,Y 458.545,Z 554.635,A -85,B 0,C 180,E1 21203.156,E2 21203.156} C_VEL
LIN {X 0,Y 466.084,Z 565.379,A -85,B 0,C 180,E1 21201.686,E2 21201.686} C_VEL
LIN {X 0,Y 477.232,Z 582.151,A -85,B 0,C 180,E1 21199.655,E2 21199.655} C_VEL
LIN {X 0,Y 482.883,Z 591.612,A -85,B 0,C 180,E1 21198.671,E2 21198.671} C_VEL
LIN {X 0,Y 477.025,Z 790.763,A -85,B 0,C 180,E1 21195.157,E2 21195.157} C_VEL
LIN {X 0,Y 474.061,Z 890.88,A -85,B 0,C 180,E1 21193.394,E2 21193.394} C_VEL
LIN {X 0,Y 472.453,Z 914.267,A -85,B 0,C 180,E1 21192.797,E2 21192.797} C_VEL
LIN {X 0,Y 470.542,Z 936.616,A -85,B 0,C 180,E1 21192.017,E2 21192.017} C_VEL
LIN {X 0,Y 468.219,Z 957.779,A -85,B 0,C 180,E1 21191.053,E2 21191.053} C_VEL
LIN {X 0,Y 465.737,Z 978.107,A -85,B 0,C 180,E1 21189.934,E2 21189.934} C_VEL
LIN {X 0,Y 462.833,Z 998.698,A -85,B 0,C 180,E1 21188.554,E2 21188.554} C_VEL
LIN {X 0,Y 459.854,Z 1018.96,A -85,B 0,C 180,E1 21186.955,E2 21186.955} C_VEL
LIN {X 0,Y 456.891,Z 1037.595,A -85,B 0,C 180,E1 21185.215,E2 21185.215} C_VEL
LIN {X 0,Y 453.779,Z 1056.767,A -85,B 0,C 180,E1 21183.145,E2 21183.145} C_VEL
LIN {X 0,Y 451.061,Z 1073.549,A -85,B 0,C 180,E1 21181.036,E2 21181.036} C_VEL
LIN {X 0,Y 448.416,Z 1090.057,A -85,B 0,C 180,E1 21178.646,E2 21178.646} C_VEL
LIN {X 0,Y 446.319,Z 1103.958,A -85,B 0,C 180,E1 21176.331,E2 21176.331} C_VEL
LIN {X 0,Y 444.296,Z 1117.804,A -85,B 0,C 180,E1 21173.614,E2 21173.614} C_VEL
LIN {X 0,Y 442.768,Z 1129.723,A -85,B 0,C 180,E1 21170.903,E2 21170.903} C_VEL
LIN {X 0,Y 441.594,Z 1140.142,A -85,B 0,C 180,E1 21168.071,E2 21168.071} C_VEL
LIN {X 0,Y 440.785,Z 1149.286,A -85,B 0,C 180,E1 21165.121,E2 21165.121} C_VEL
LIN {X 0,Y 440.319,Z 1155.955,A -85,B 0,C 180,E1 21162.458,E2 21162.458} C_VEL
LIN {X 0,Y 440.051,Z 1161.81,A -85,B 0,C 180,E1 21159.547,E2 21159.547} C_VEL
LIN {X 0,Y 439.937,Z 1165.8,A -85,B 0,C 180,E1 21156.787,E2 21156.787} C_VEL
LIN {X 0,Y 439.91,Z 1168.632,A -85,B 0,C 180,E1 21153.91,E2 21153.91} C_VEL
LIN {X 0,Y 439.894,Z 1169.826,A -85,B 0,C 180,E1 21151.042,E2 21151.042} C_VEL
LIN {X 0,Y 439.906,Z 1169.735,A -85,B 0,C 180,E1 21148.437,E2 21148.437} C_VEL
LIN {X 0,Y 439.911,Z 1168.068,A -85,B 0,C 180,E1 21145.437,E2 21145.437} C_VEL
LIN {X 0,Y 439.934,Z 1165.319,A -85,B 0,C 180,E1 21142.819,E2 21142.819} C_VEL
LIN {X 0,Y 440.086,Z 1160.589,A -85,B 0,C 180,E1 21139.792,E2 21139.792} C_VEL
LIN {X 0,Y 440.369,Z 1155.043,A -85,B 0,C 180,E1 21137.143,E2 21137.143} C_VEL
LIN {X 0,Y 440.989,Z 1146.767,A -85,B 0,C 180,E1 21134.014,E2 21134.014} C_VEL
LIN {X 0,Y 441.849,Z 1137.85,A -85,B 0,C 180,E1 21131.256,E2 21131.256} C_VEL
LIN {X 0,Y 443.136,Z 1126.66,A -85,B 0,C 180,E1 21128.372,E2 21128.372} C_VEL
LIN {X 0,Y 444.766,Z 1114.623,A -85,B 0,C 180,E1 21125.707,E2 21125.707} C_VEL
LIN {X 0,Y 446.662,Z 1101.616,A -85,B 0,C 180,E1 21123.26,E2 21123.26} C_VEL
LIN {X 0,Y 449.01,Z 1086.496,A -85,B 0,C 180,E1 21120.797,E2 21120.797} C_VEL
LIN {X 0,Y 451.661,Z 1069.74,A -85,B 0,C 180,E1 21118.461,E2 21118.461} C_VEL
LIN {X 0,Y 454.731,Z 1050.991,A -85,B 0,C 180,E1 21116.2,E2 21116.2} C_VEL
LIN {X 0,Y 457.54,Z 1033.536,A -85,B 0,C 180,E1 21114.382,E2 21114.382} C_VEL
LIN {X 0,Y 460.683,Z 1013.284,A -85,B 0,C 180,E1 21112.575,E2 21112.575} C_VEL
LIN {X 0,Y 463.669,Z 993.248,A -85,B 0,C 180,E1 21111.053,E2 21111.053} C_VEL
LIN {X 0,Y 466.49,Z 971.904,A -85,B 0,C 180,E1 21109.706,E2 21109.706} C_VEL
LIN {X 0,Y 469.04,Z 950.757,A -85,B 0,C 180,E1 21108.595,E2 21108.595} C_VEL
LIN {X 0,Y 471.267,Z 928.34,A -85,B 0,C 180,E1 21107.673,E2 21107.673} C_VEL
LIN {X 0,Y 473.205,Z 904.792,A -85,B 0,C 180,E1 21106.935,E2 21106.935} C_VEL
LIN {X 0,Y 474.397,Z 882.917,A -85,B 0,C 180,E1 21106.451,E2 21106.451} C_VEL
LIN {X 0,Y 480.078,Z 684.212,A -85,B 0,C 180,E1 21102.972,E2 21102.972} C_VEL
LIN {X 0,Y 482.792,Z 591.141,A -85,B 0,C 180,E1 21101.309,E2 21101.309} C_VEL
LIN {X 0,Y 471.928,Z 574.13,A -85,B 0,C 180,E1 21099.405,E2 21099.405} C_VEL
LIN {X 0,Y 460.792,Z 557.672,A -85,B 0,C 180,E1 21097.296,E2 21097.296} C_VEL
LIN {X 0,Y 452.226,Z 546.057,A -85,B 0,C 180,E1 21095.555,E2 21095.555} C_VEL
LIN {X 0,Y 449.414,Z 542.22,A -85,B 0,C 180,E1 21094.951,E2 21094.951} C_VEL
LIN {X 0,Y 445.848,Z 537.318,A -85,B 0,C 180,E1 21094.154,E2 21094.154} C_VEL
LIN {X 0,Y 443.929,Z 533.533,A -85,B 0,C 180,E1 21093.32,E2 21093.32} C_VEL
LIN {X 0,Y 441.452,Z 529.437,A -85,B 0,C 180,E1 21092.311,E2 21092.311} C_VEL
LIN {X 0,Y 441.161,Z 528.092,A -85,B 0,C 180,E1 21092.028,E2 21092.028} C_VEL
LIN {X 0,Y 441.17,Z 528.056,A -85,B 0,C 180,E1 21088.273,E2 21088.273} C_VEL
LIN {X 0,Y 441.192,Z 528.048,A -85,B 0,C 180,E1 21084.644,E2 21084.644} C_VEL
LIN {X 0,Y 441.197,Z 528.089,A -85,B 0,C 180,E1 21080.842,E2 21080.842} C_VEL
LIN {X 0,Y 441.179,Z 528.043,A -85,B 0,C 180,E1 21076.999,E2 21076.999} C_VEL
LIN {X 0,Y 441.181,Z 528.083,A -85,B 0,C 180,E1 21073.232,E2 21073.232} C_VEL
LIN {X 0,Y 441.188,Z 528.057,A -85,B 0,C 180,E1 21069.391,E2 21069.391} C_VEL
LIN {X 0,Y 441.185,Z 528.079,A -85,B 0,C 180,E1 21065.723,E2 21065.723} C_VEL
LIN {X 0,Y 441.186,Z 528.081,A -85,B 0,C 180,E1 21061.902,E2 21061.902} C_VEL
LIN {X 0,Y 441.193,Z 528.08,A -85,B 0,C 180,E1 21058.182,E2 21058.182} C_VEL
LIN {X 0,Y 441.192,Z 528.078,A -85,B 0,C 180,E1 21054.407,E2 21054.407} C_VEL
LIN {X 0,Y 441.177,Z 528.056,A -85,B 0,C 180,E1 21050.74,E2 21050.74} C_VEL
LIN {X 0,Y 441.167,Z 528.08,A -85,B 0,C 180,E1 21047.034,E2 21047.034} C_VEL
LIN {X 0,Y 441.184,Z 528.046,A -85,B 0,C 180,E1 21043.408,E2 21043.408} C_VEL
LIN {X 0,Y 441.2,Z 528.089,A -85,B 0,C 180,E1 21039.574,E2 21039.574} C_VEL
LIN {X 0,Y 441.167,Z 528.045,A -85,B 0,C 180,E1 21035.924,E2 21035.924} C_VEL
LIN {X 0,Y 441.15,Z 528.084,A -85,B 0,C 180,E1 21032.314,E2 21032.314} C_VEL
LIN {X 0,Y 441.172,Z 528.073,A -85,B 0,C 180,E1 21028.697,E2 21028.697} C_VEL
LIN {X 0,Y 441.172,Z 528.188,A -85,B 0,C 180,E1 21026.427,E2 21026.427} C_VEL
LIN {X 0,Y 442.239,Z 531.223,A -85,B 0,C 180,E1 21026.13,E2 21026.13} C_VEL
LIN {X 0,Y 444.762,Z 533.802,A -85,B 0,C 180,E1 21025.57,E2 21025.57} C_VEL
LIN {X 0,Y 445.866,Z 534.72,A -85,B 0,C 180,E1 21025.336,E2 21025.336} C_VEL
LIN {X 0,Y 448.258,Z 538.487,A -85,B 0,C 180,E1 21024.788,E2 21024.788} C_VEL
LIN {X 0,Y 450.521,Z 540.799,A -85,B 0,C 180,E1 21024.316,E2 21024.316} C_VEL
LIN {X 0,Y 453.705,Z 545.005,A -85,B 0,C 180,E1 21023.643,E2 21023.643} C_VEL
LIN {X 0,Y 455.408,Z 547.213,A -85,B 0,C 180,E1 21023.292,E2 21023.292} C_VEL
LIN {X 0,Y 462.925,Z 556.845,A -85,B 0,C 180,E1 21021.81,E2 21021.81} C_VEL
LIN {X 0,Y 475.177,Z 573.689,A -85,B 0,C 180,E1 21019.563,E2 21019.563} C_VEL
LIN {X 0,Y 482.689,Z 584.861,A -85,B 0,C 180,E1 21018.27,E2 21018.27} C_VEL
LIN {X 0,Y 476.363,Z 797.916,A -85,B 0,C 180,E1 21014.514,E2 21014.514} C_VEL
LIN {X 0,Y 475.807,Z 817.75,A -85,B 0,C 180,E1 21014.169,E2 21014.169} C_VEL
LIN {X 0,Y 474.874,Z 825.449,A -85,B 0,C 180,E1 21014.12,E2 21014.12} C_VEL
LIN {X 0,Y 469.817,Z 846.036,A -85,B 0,C 180,E1 21014.294,E2 21014.294} C_VEL
LIN {X 0,Y 469.076,Z 852.641,A -85,B 0,C 180,E1 21014.242,E2 21014.242} C_VEL
LIN {X 0,Y 467.886,Z 875.575,A -85,B 0,C 180,E1 21013.748,E2 21013.748} C_VEL
LIN {X 0,Y 466.217,Z 897.569,A -85,B 0,C 180,E1 21013.089,E2 21013.089} C_VEL
LIN {X 0,Y 464.056,Z 918.72,A -85,B 0,C 180,E1 21012.241,E2 21012.241} C_VEL
LIN {X 0,Y 461.402,Z 940.893,A -85,B 0,C 180,E1 21011.124,E2 21011.124} C_VEL
LIN {X 0,Y 458.709,Z 960.18,A -85,B 0,C 180,E1 21009.928,E2 21009.928} C_VEL
LIN {X 0,Y 455.533,Z 980.863,A -85,B 0,C 180,E1 21008.402,E2 21008.402} C_VEL
LIN {X 0,Y 452.418,Z 999.25,A -85,B 0,C 180,E1 21006.793,E2 21006.793} C_VEL
LIN {X 0,Y 448.91,Z 1018.995,A -85,B 0,C 180,E1 21004.764,E2 21004.764} C_VEL
LIN {X 0,Y 445.816,Z 1036.06,A -85,B 0,C 180,E1 21002.719,E2 21002.719} C_VEL
LIN {X 0,Y 442.726,Z 1052.669,A -85,B 0,C 180,E1 21000.391,E2 21000.391} C_VEL
LIN {X 0,Y 440.023,Z 1067.995,A -85,B 0,C 180,E1 20997.911,E2 20997.911} C_VEL
LIN {X 0,Y 437.765,Z 1081.115,A -85,B 0,C 180,E1 20995.43,E2 20995.43} C_VEL
LIN {X 0,Y 435.646,Z 1094.957,A -85,B 0,C 180,E1 20992.395,E2 20992.395} C_VEL
LIN {X 0,Y 434.252,Z 1105.757,A -85,B 0,C 180,E1 20989.644,E2 20989.644} C_VEL
LIN {X 0,Y 433.204,Z 1115.417,A -85,B 0,C 180,E1 20986.696,E2 20986.696} C_VEL
LIN {X 0,Y 432.545,Z 1123.403,A -85,B 0,C 180,E1 20983.774,E2 20983.774} C_VEL
LIN {X 0,Y 432.17,Z 1129.741,A -85,B 0,C 180,E1 20980.801,E2 20980.801} C_VEL
LIN {X 0,Y 431.988,Z 1134.622,A -85,B 0,C 180,E1 20977.849,E2 20977.849} C_VEL
LIN {X 0,Y 431.917,Z 1137.802,A -85,B 0,C 180,E1 20974.914,E2 20974.914} C_VEL
LIN {X 0,Y 431.91,Z 1139.572,A -85,B 0,C 180,E1 20972.123,E2 20972.123} C_VEL
LIN {X 0,Y 431.884,Z 1139.879,A -85,B 0,C 180,E1 20969.204,E2 20969.204} C_VEL
LIN {X 0,Y 431.886,Z 1139.007,A -85,B 0,C 180,E1 20966.682,E2 20966.682} C_VEL
LIN {X 0,Y 431.939,Z 1136.492,A -85,B 0,C 180,E1 20963.621,E2 20963.621} C_VEL
LIN {X 0,Y 432.038,Z 1132.912,A -85,B 0,C 180,E1 20960.946,E2 20960.946} C_VEL
LIN {X 0,Y 432.296,Z 1127.267,A -85,B 0,C 180,E1 20957.85,E2 20957.85} C_VEL
LIN {X 0,Y 432.768,Z 1120.461,A -85,B 0,C 180,E1 20955.004,E2 20955.004} C_VEL
LIN {X 0,Y 433.644,Z 1111.207,A -85,B 0,C 180,E1 20951.864,E2 20951.864} C_VEL
LIN {X 0,Y 434.796,Z 1101.452,A -85,B 0,C 180,E1 20949.119,E2 20949.119} C_VEL
LIN {X 0,Y 436.567,Z 1088.68,A -85,B 0,C 180,E1 20946.085,E2 20946.085} C_VEL
LIN {X 0,Y 438.642,Z 1076.027,A -85,B 0,C 180,E1 20943.464,E2 20943.464} C_VEL
LIN {X 0,Y 441.054,Z 1061.932,A -85,B 0,C 180,E1 20940.979,E2 20940.979} C_VEL
LIN {X 0,Y 444.025,Z 1045.75,A -85,B 0,C 180,E1 20938.505,E2 20938.505} C_VEL
LIN {X 0,Y 446.972,Z 1029.596,A -85,B 0,C 180,E1 20936.383,E2 20936.383} C_VEL
LIN {X 0,Y 450.372,Z 1010.931,A -85,B 0,C 180,E1 20934.276,E2 20934.276} C_VEL
LIN {X 0,Y 453.42,Z 993.551,A -85,B 0,C 180,E1 20932.59,E2 20932.59} C_VEL
LIN {X 0,Y 456.712,Z 973.231,A -85,B 0,C 180,E1 20930.913,E2 20930.913} C_VEL
LIN {X 0,Y 459.746,Z 953.215,A -85,B 0,C 180,E1 20929.52,E2 20929.52} C_VEL
LIN {X 0,Y 462.479,Z 932.402,A -85,B 0,C 180,E1 20928.333,E2 20928.333} C_VEL
LIN {X 0,Y 464.898,Z 911.49,A -85,B 0,C 180,E1 20927.353,E2 20927.353} C_VEL
LIN {X 0,Y 466.886,Z 889.206,A -85,B 0,C 180,E1 20926.549,E2 20926.549} C_VEL
LIN {X 0,Y 468.441,Z 867.234,A -85,B 0,C 180,E1 20925.955,E2 20925.955} C_VEL
LIN {X 0,Y 470.377,Z 809.002,A -85,B 0,C 180,E1 20924.902,E2 20924.902} C_VEL
LIN {X 0,Y 477.03,Z 597.168,A -85,B 0,C 180,E1 20921.138,E2 20921.138} C_VEL
LIN {X 0,Y 477.19,Z 588.404,A -85,B 0,C 180,E1 20920.963,E2 20920.963} C_VEL
LIN {X 0,Y 465.457,Z 571.497,A -85,B 0,C 180,E1 20918.848,E2 20918.848} C_VEL
LIN {X 0,Y 454.8,Z 557.22,A -85,B 0,C 180,E1 20916.765,E2 20916.765} C_VEL
LIN {X 0,Y 450.092,Z 551.293,A -85,B 0,C 180,E1 20915.789,E2 20915.789} C_VEL
LIN {X 0,Y 446.27,Z 546.359,A -85,B 0,C 180,E1 20914.96,E2 20914.96} C_VEL
LIN {X 0,Y 443.026,Z 542.169,A -85,B 0,C 180,E1 20914.231,E2 20914.231} C_VEL
LIN {X 0,Y 441.904,Z 540.871,A -85,B 0,C 180,E1 20913.978,E2 20913.978} C_VEL
LIN {X 0,Y 438.94,Z 537.563,A -85,B 0,C 180,E1 20913.297,E2 20913.297} C_VEL
LIN {X 0,Y 437.555,Z 535.197,A -85,B 0,C 180,E1 20912.947,E2 20912.947} C_VEL
LIN {X 0,Y 434.718,Z 532.856,A -85,B 0,C 180,E1 20912.288,E2 20912.288} C_VEL
LIN {X 0,Y 433.353,Z 529.928,A -85,B 0,C 180,E1 20911.909,E2 20911.909} C_VEL
LIN {X 0,Y 433.203,Z 529.089,A -85,B 0,C 180,E1 20911.836,E2 20911.836} C_VEL
LIN {X 0,Y 433.21,Z 529.052,A -85,B 0,C 180,E1 20908.089,E2 20908.089} C_VEL
LIN {X 0,Y 433.247,Z 529.037,A -85,B 0,C 180,E1 20904.4,E2 20904.4} C_VEL
LIN {X 0,Y 433.252,Z 529.079,A -85,B 0,C 180,E1 20900.677,E2 20900.677} C_VEL
LIN {X 0,Y 433.222,Z 529.03,A -85,B 0,C 180,E1 20896.906,E2 20896.906} C_VEL
LIN {X 0,Y 433.226,Z 529.083,A -85,B 0,C 180,E1 20893.107,E2 20893.107} C_VEL
LIN {X 0,Y 433.242,Z 529.077,A -85,B 0,C 180,E1 20889.297,E2 20889.297} C_VEL
LIN {X 0,Y 433.257,Z 529.071,A -85,B 0,C 180,E1 20885.562,E2 20885.562} C_VEL
LIN {X 0,Y 433.255,Z 529.069,A -85,B 0,C 180,E1 20881.719,E2 20881.719} C_VEL
LIN {X 0,Y 433.247,Z 529.071,A -85,B 0,C 180,E1 20878.016,E2 20878.016} C_VEL
LIN {X 0,Y 433.244,Z 529.069,A -85,B 0,C 180,E1 20874.172,E2 20874.172} C_VEL
LIN {X 0,Y 433.251,Z 529.05,A -85,B 0,C 180,E1 20870.436,E2 20870.436} C_VEL
LIN {X 0,Y 433.242,Z 529.062,A -85,B 0,C 180,E1 20866.657,E2 20866.657} C_VEL
LIN {X 0,Y 433.236,Z 529.035,A -85,B 0,C 180,E1 20862.818,E2 20862.818} C_VEL
LIN {X 0,Y 433.256,Z 529.083,A -85,B 0,C 180,E1 20859.041,E2 20859.041} C_VEL
LIN {X 0,Y 433.254,Z 529.045,A -85,B 0,C 180,E1 20855.165,E2 20855.165} C_VEL
LIN {X 0,Y 433.252,Z 529.042,A -85,B 0,C 180,E1 20851.464,E2 20851.464} C_VEL
LIN {X 0,Y 433.276,Z 529.263,A -85,B 0,C 180,E1 20849.402,E2 20849.402} C_VEL
LIN {X 0,Y 434.561,Z 532.566,A -85,B 0,C 180,E1 20848.669,E2 20848.669} C_VEL
LIN {X 0,Y 435.956,Z 534.165,A -85,B 0,C 180,E1 20848.164,E2 20848.164} C_VEL
LIN {X 0,Y 437.503,Z 537.514,A -85,B 0,C 180,E1 20847.478,E2 20847.478} C_VEL
LIN {X 0,Y 440.04,Z 540.689,A -85,B 0,C 180,E1 20846.876,E2 20846.876} C_VEL
LIN {X 0,Y 444.217,Z 546.134,A -85,B 0,C 180,E1 20845.913,E2 20845.913} C_VEL
LIN {X 0,Y 454.165,Z 559.583,A -85,B 0,C 180,E1 20843.765,E2 20843.765} C_VEL
LIN {X 0,Y 466.403,Z 577.51,A -85,B 0,C 180,E1 20841.345,E2 20841.345} C_VEL
LIN {X 0,Y 477.47,Z 595.033,A -85,B 0,C 180,E1 20839.331,E2 20839.331} C_VEL
LIN {X 0,Y 471.361,Z 791.244,A -85,B 0,C 180,E1 20835.838,E2 20835.838} C_VEL
LIN {X 0,Y 468.247,Z 890.59,A -85,B 0,C 180,E1 20834.071,E2 20834.071} C_VEL
LIN {X 0,Y 466.543,Z 914.1,A -85,B 0,C 180,E1 20833.467,E2 20833.467} C_VEL
